LIN {X 0,Y 329.805,Z 667.304,A -85,B 0,C 180,E1 16241.947,E2 16241.947} C_VEL
LIN {X 0,Y 329.564,Z 671.373,A -85,B 0,C 180,E1 16242.444,E2 16242.444} C_VEL
LIN {X 0,Y 319.657,Z 703.267,A -85,B 0,C 180,E1 16245.4,E2 16245.4} C_VEL
LIN {X 0,Y 308.366,Z 732.75,A -85,B 0,C 180,E1 16249.353,E2 16249.353} C_VEL
LIN {X 0,Y 296.702,Z 759.051,A -85,B 0,C 180,E1 16254.413,E2 16254.413} C_VEL
LIN {X 0,Y 286.049,Z 781.446,A -85,B 0,C 180,E1 16260.671,E2 16260.671} C_VEL
LIN {X 0,Y 278.02,Z 798.479,A -85,B 0,C 180,E1 16267.777,E2 16267.777} C_VEL
LIN {X 0,Y 273.133,Z 810.385,A -85,B 0,C 180,E1 16275.599,E2 16275.599} C_VEL
LIN {X 0,Y 271.089,Z 816.889,A -85,B 0,C 180,E1 16283.586,E2 16283.586} C_VEL
LIN {X 0,Y 270.872,Z 818.496,A -85,B 0,C 180,E1 16289.999,E2 16289.999} C_VEL
LIN {X 0,Y 271.134,Z 816.829,A -85,B 0,C 180,E1 16296.412,E2 16296.412} C_VEL
LIN {X 0,Y 273.229,Z 810.161,A -85,B 0,C 180,E1 16304.483,E2 16304.483} C_VEL
LIN {X 0,Y 278.223,Z 797.96,A -85,B 0,C 180,E1 16312.391,E2 16312.391} C_VEL
LIN {X 0,Y 286.286,Z 780.835,A -85,B 0,C 180,E1 16319.419,E2 16319.419} C_VEL
LIN {X 0,Y 296.961,Z 758.345,A -85,B 0,C 180,E1 16325.639,E2 16325.639} C_VEL
LIN {X 0,Y 308.651,Z 731.826,A -85,B 0,C 180,E1 16330.691,E2 16330.691} C_VEL
LIN {X 0,Y 320.1,Z 701.772,A -85,B 0,C 180,E1 16334.662,E2 16334.662} C_VEL
LIN {X 0,Y 330.02,Z 668.599,A -85,B 0,C 180,E1 16337.711,E2 16337.711} C_VEL
LIN {X 0,Y 322.594,Z 643.397,A -85,B 0,C 180,E1 16342.404,E2 16342.404} C_VEL
LIN {X 0,Y 312.412,Z 620.496,A -85,B 0,C 180,E1 16347.568,E2 16347.568} C_VEL
LIN {X 0,Y 300.457,Z 599.556,A -85,B 0,C 180,E1 16353.739,E2 16353.739} C_VEL
LIN {X 0,Y 290.832,Z 585.901,A -85,B 0,C 180,E1 16359.592,E2 16359.592} C_VEL
LIN {X 0,Y 286.331,Z 579.387,A -85,B 0,C 180,E1 16363.177,E2 16363.177} C_VEL
LIN {X 0,Y 282.314,Z 573.377,A -85,B 0,C 180,E1 16367.516,E2 16367.516} C_VEL
LIN {X 0,Y 278.321,Z 569.305,A -85,B 0,C 180,E1 16376.882,E2 16376.882} C_VEL
LIN {X 0,Y 279.401,Z 570.647,A -85,B 0,C 180,E1 16383.301,E2 16383.301} C_VEL
LIN {X 0,Y 282.503,Z 573.483,A -85,B 0,C 180,E1 16388.281,E2 16388.281} C_VEL
LIN {X 0,Y 286.101,Z 579.139,A -85,B 0,C 180,E1 16392.221,E2 16392.221} C_VEL
LIN {X 0,Y 287.999,Z 581.762,A -85,B 0,C 180,E1 16393.861,E2 16393.861} C_VEL
LIN {X 0,Y 293.39,Z 589.45,A -85,B 0,C 180,E1 16397.745,E2 16397.745} C_VEL
LIN {X 0,Y 301.462,Z 601.319,A -85,B 0,C 180,E1 16402.418,E2 16402.418} C_VEL
LIN {X 0,Y 313.146,Z 621.425,A -85,B 0,C 180,E1 16408.222,E2 16408.222} C_VEL
LIN {X 0,Y 323.586,Z 644.854,A -85,B 0,C 180,E1 16413.27,E2 16413.27} C_VEL
LIN {X 0,Y 331.263,Z 670.261,A -85,B 0,C 180,E1 16417.717,E2 16417.717} C_VEL
LIN {X 0,Y 320.897,Z 707.285,A -85,B 0,C 180,E1 16420.726,E2 16420.726} C_VEL
LIN {X 0,Y 309.149,Z 741.143,A -85,B 0,C 180,E1 16424.755,E2 16424.755} C_VEL
LIN {X 0,Y 297.16,Z 771.177,A -85,B 0,C 180,E1 16429.837,E2 16429.837} C_VEL
LIN {X 0,Y 286.1,Z 797.759,A -85,B 0,C 180,E1 16436.244,E2 16436.244} C_VEL
LIN {X 0,Y 277.977,Z 818.25,A -85,B 0,C 180,E1 16443.299,E2 16443.299} C_VEL
LIN {X 0,Y 272.92,Z 834.265,A -85,B 0,C 180,E1 16451.399,E2 16451.399} C_VEL
LIN {X 0,Y 270.979,Z 843.701,A -85,B 0,C 180,E1 16458.924,E2 16458.924} C_VEL
LIN {X 0,Y 270.477,Z 848.401,A -85,B 0,C 180,E1 16466.792,E2 16466.792} C_VEL
LIN {X 0,Y 270.551,Z 848.411,A -85,B 0,C 180,E1 16473.209,E2 16473.209} C_VEL
LIN {X 0,Y 270.986,Z 843.71,A -85,B 0,C 180,E1 16481.085,E2 16481.085} C_VEL
LIN {X 0,Y 273.236,Z 832.973,A -85,B 0,C 180,E1 16489.419,E2 16489.419} C_VEL
LIN {X 0,Y 278.709,Z 816.254,A -85,B 0,C 180,E1 16497.501,E2 16497.501} C_VEL
LIN {X 0,Y 287.215,Z 795.052,A -85,B 0,C 180,E1 16504.52,E2 16504.52} C_VEL
LIN {X 0,Y 297.881,Z 769.444,A -85,B 0,C 180,E1 16510.524,E2 16510.524} C_VEL
LIN {X 0,Y 310.009,Z 738.891,A -85,B 0,C 180,E1 16515.584,E2 16515.584} C_VEL
LIN {X 0,Y 321.936,Z 704.311,A -85,B 0,C 180,E1 16519.579,E2 16519.579} C_VEL
LIN {X 0,Y 331.184,Z 669.723,A -85,B 0,C 180,E1 16522.393,E2 16522.393} C_VEL
LIN {X 0,Y 323.663,Z 644.953,A -85,B 0,C 180,E1 16526.739,E2 16526.739} C_VEL
LIN {X 0,Y 315.532,Z 626.221,A -85,B 0,C 180,E1 16530.694,E2 16530.694} C_VEL
LIN {X 0,Y 311.88,Z 623.31,A -85,B 0,C 180,E1 16532.061,E2 16532.061} C_VEL
LIN {X 0,Y 305.951,Z 620.829,A -85,B 0,C 180,E1 16534.268,E2 16534.268} C_VEL
LIN {X 0,Y 305.532,Z 620.05,A -85,B 0,C 180,E1 16534.493,E2 16534.493} C_VEL
LIN {X 0,Y 295.869,Z 603.458,A -85,B 0,C 180,E1 16539.989,E2 16539.989} C_VEL
LIN {X 0,Y 288.98,Z 593.047,A -85,B 0,C 180,E1 16544.626,E2 16544.626} C_VEL
LIN {X 0,Y 284.687,Z 586.778,A -85,B 0,C 180,E1 16548.302,E2 16548.302} C_VEL
LIN {X 0,Y 281.092,Z 580.621,A -85,B 0,C 180,E1 16552.576,E2 16552.576} C_VEL
LIN {X 0,Y 277.764,Z 577.392,A -85,B 0,C 180,E1 16559.999,E2 16559.999} C_VEL
LIN {X 0,Y 280.92,Z 580.502,A -85,B 0,C 180,E1 16571.484,E2 16571.484} C_VEL
LIN {X 0,Y 284.724,Z 586.915,A -85,B 0,C 180,E1 16576.024,E2 16576.024} C_VEL
LIN {X 0,Y 287.489,Z 591.3,A -85,B 0,C 180,E1 16578.532,E2 16578.532} C_VEL
LIN {X 0,Y 291.493,Z 597.021,A -85,B 0,C 180,E1 16581.518,E2 16581.518} C_VEL
LIN {X 0,Y 299.641,Z 609.825,A -85,B 0,C 180,E1 16586.641,E2 16586.641} C_VEL
LIN {X 0,Y 309.655,Z 628.692,A -85,B 0,C 180,E1 16592.224,E2 16592.224} C_VEL
LIN {X 0,Y 319.03,Z 652.103,A -85,B 0,C 180,E1 16597.568,E2 16597.568} C_VEL
LIN {X 0,Y 324.068,Z 672.936,A -85,B 0,C 180,E1 16601.485,E2 16601.485} C_VEL
LIN {X 0,Y 313.257,Z 706.117,A -85,B 0,C 180,E1 16604.642,E2 16604.642} C_VEL
LIN {X 0,Y 300.569,Z 737.537,A -85,B 0,C 180,E1 16609.072,E2 16609.072} C_VEL
LIN {X 0,Y 287.912,Z 764.286,A -85,B 0,C 180,E1 16614.657,E2 16614.657} C_VEL
LIN {X 0,Y 277.608,Z 784.776,A -85,B 0,C 180,E1 16620.916,E2 16620.916} C_VEL
LIN {X 0,Y 269.758,Z 800.788,A -85,B 0,C 180,E1 16628.163,E2 16628.163} C_VEL
LIN {X 0,Y 264.991,Z 811.989,A -85,B 0,C 180,E1 16636.223,E2 16636.223} C_VEL
LIN {X 0,Y 263.217,Z 817.334,A -85,B 0,C 180,E1 16643.393,E2 16643.393} C_VEL
LIN {X 0,Y 262.982,Z 818.939,A -85,B 0,C 180,E1 16649.999,E2 16649.999} C_VEL
LIN {X 0,Y 263.262,Z 817.274,A -85,B 0,C 180,E1 16656.604,E2 16656.604} C_VEL
LIN {X 0,Y 265.572,Z 810.523,A -85,B 0,C 180,E1 16664.991,E2 16664.991} C_VEL
LIN {X 0,Y 270.838,Z 798.417,A -85,B 0,C 180,E1 16673.036,E2 16673.036} C_VEL
LIN {X 0,Y 279.651,Z 780.628,A -85,B 0,C 180,E1 16680.455,E2 16680.455} C_VEL
LIN {X 0,Y 290.989,Z 757.949,A -85,B 0,C 180,E1 16686.752,E2 16686.752} C_VEL
LIN {X 0,Y 303.284,Z 730.998,A -85,B 0,C 180,E1 16691.888,E2 16691.888} C_VEL
LIN {X 0,Y 315.639,Z 699.335,A -85,B 0,C 180,E1 16696.014,E2 16696.014} C_VEL
LIN {X 0,Y 324.096,Z 671.324,A -85,B 0,C 180,E1 16698.609,E2 16698.609} C_VEL
LIN {X 0,Y 316.842,Z 645.653,A -85,B 0,C 180,E1 16703.659,E2 16703.659} C_VEL
LIN {X 0,Y 306.787,Z 622.65,A -85,B 0,C 180,E1 16709.227,E2 16709.227} C_VEL
LIN {X 0,Y 296.838,Z 605.304,A -85,B 0,C 180,E1 16714.815,E2 16714.815} C_VEL
LIN {X 0,Y 288.776,Z 593.022,A -85,B 0,C 180,E1 16720.224,E2 16720.224} C_VEL
LIN {X 0,Y 284.732,Z 586.895,A -85,B 0,C 180,E1 16723.692,E2 16723.692} C_VEL
LIN {X 0,Y 280.49,Z 580.156,A -85,B 0,C 180,E1 16728.693,E2 16728.693} C_VEL
LIN {X 0,Y 277.532,Z 577.075,A -85,B 0,C 180,E1 16740.001,E2 16740.001} C_VEL
LIN {X 0,Y 281.204,Z 581.256,A -85,B 0,C 180,E1 16747.93,E2 16747.93} C_VEL
LIN {X 0,Y 285.33,Z 587.159,A -85,B 0,C 180,E1 16752.428,E2 16752.428} C_VEL
LIN {X 0,Y 292.338,Z 598.219,A -85,B 0,C 180,E1 16757.908,E2 16757.908} C_VEL
LIN {X 0,Y 301.675,Z 612.953,A -85,B 0,C 180,E1 16763.475,E2 16763.475} C_VEL
LIN {X 0,Y 312.271,Z 633.888,A -85,B 0,C 180,E1 16769.112,E2 16769.112} C_VEL
LIN {X 0,Y 321.29,Z 657.275,A -85,B 0,C 180,E1 16774.026,E2 16774.026} C_VEL
LIN {X 0,Y 325.329,Z 673.89,A -85,B 0,C 180,E1 16776.917,E2 16776.917} C_VEL
LIN {X 0,Y 314.607,Z 709.827,A -85,B 0,C 180,E1 16779.93,E2 16779.93} C_VEL
LIN {X 0,Y 302.053,Z 744.114,A -85,B 0,C 180,E1 16784.161,E2 16784.161} C_VEL
LIN {X 0,Y 289.556,Z 773.856,A -85,B 0,C 180,E1 16789.452,E2 16789.452} C_VEL
LIN {X 0,Y 278.152,Z 799.801,A -85,B 0,C 180,E1 16796.088,E2 16796.088} C_VEL
LIN {X 0,Y 269.934,Z 819.61,A -85,B 0,C 180,E1 16803.339,E2 16803.339} C_VEL
LIN {X 0,Y 265.234,Z 833.802,A -85,B 0,C 180,E1 16810.839,E2 16810.839} C_VEL
LIN {X 0,Y 263.211,Z 842.567,A -85,B 0,C 180,E1 16817.91,E2 16817.91} C_VEL
LIN {X 0,Y 262.653,Z 846.617,A -85,B 0,C 180,E1 16823.38,E2 16823.38} C_VEL
LIN {X 0,Y 262.814,Z 848.446,A -85,B 0,C 180,E1 16830.001,E2 16830.001} C_VEL
LIN {X 0,Y 262.769,Z 845.695,A -85,B 0,C 180,E1 16838.283,E2 16838.283} C_VEL
LIN {X 0,Y 264.269,Z 837.438,A -85,B 0,C 180,E1 16846.647,E2 16846.647} C_VEL
LIN {X 0,Y 268.842,Z 822.671,A -85,B 0,C 180,E1 16855.298,E2 16855.298} C_VEL
LIN {X 0,Y 277.086,Z 802.365,A -85,B 0,C 180,E1 16863.122,E2 16863.122} C_VEL
LIN {X 0,Y 287.795,Z 777.785,A -85,B 0,C 180,E1 16869.701,E2 16869.701} C_VEL
LIN {X 0,Y 299.815,Z 749.596,A -85,B 0,C 180,E1 16875.012,E2 16875.012} C_VEL
LIN {X 0,Y 311.995,Z 717.953,A -85,B 0,C 180,E1 16879.198,E2 16879.198} C_VEL
LIN {X 0,Y 322.866,Z 683.592,A -85,B 0,C 180,E1 16882.382,E2 16882.382} C_VEL
LIN {X 0,Y 325.391,Z 672.786,A -85,B 0,C 180,E1 16883.238,E2 16883.238} C_VEL
LIN {X 0,Y 318.483,Z 648.794,A -85,B 0,C 180,E1 16887.646,E2 16887.646} C_VEL
LIN {X 0,Y 307.903,Z 624.559,A -85,B 0,C 180,E1 16893.242,E2 16893.242} C_VEL
LIN {X 0,Y 305.532,Z 620.05,A -85,B 0,C 180,E1 16894.493,E2 16894.493} C_VEL
LIN {X 0,Y 301.126,Z 615.255,A -85,B 0,C 180,E1 16896.629,E2 16896.629} C_VEL
LIN {X 0,Y 293.286,Z 610.348,A -85,B 0,C 180,E1 16900.537,E2 16900.537} C_VEL
LIN {X 0,Y 286.858,Z 600.102,A -85,B 0,C 180,E1 16905.286,E2 16905.286} C_VEL
LIN {X 0,Y 283.021,Z 594.198,A -85,B 0,C 180,E1 16908.818,E2 16908.818} C_VEL
LIN {X 0,Y 279.274,Z 587.733,A -85,B 0,C 180,E1 16913.775,E2 16913.775} C_VEL
LIN {X 0,Y 276.799,Z 585.255,A -85,B 0,C 180,E1 16919.999,E2 16919.999} C_VEL
LIN {X 0,Y 279.653,Z 588.2,A -85,B 0,C 180,E1 16931.09,E2 16931.09} C_VEL
LIN {X 0,Y 283.599,Z 594.784,A -85,B 0,C 180,E1 16936.034,E2 16936.034} C_VEL
LIN {X 0,Y 289.739,Z 604.964,A -85,B 0,C 180,E1 16941.354,E2 16941.354} C_VEL
LIN {X 0,Y 298.315,Z 619.221,A -85,B 0,C 180,E1 16947.075,E2 16947.075} C_VEL
LIN {X 0,Y 308.334,Z 640.87,A -85,B 0,C 180,E1 16953.193,E2 16953.193} C_VEL
LIN {X 0,Y 316.21,Z 664.666,A -85,B 0,C 180,E1 16958.492,E2 16958.492} C_VEL
LIN {X 0,Y 318.119,Z 676.365,A -85,B 0,C 180,E1 16960.637,E2 16960.637} C_VEL
LIN {X 0,Y 306.215,Z 710.801,A -85,B 0,C 180,E1 16964.082,E2 16964.082} C_VEL
LIN {X 0,Y 293.721,Z 739.941,A -85,B 0,C 180,E1 16968.404,E2 16968.404} C_VEL
LIN {X 0,Y 281.094,Z 765.428,A -85,B 0,C 180,E1 16973.889,E2 16973.889} C_VEL
LIN {X 0,Y 269.837,Z 786.779,A -85,B 0,C 180,E1 16980.676,E2 16980.676} C_VEL
LIN {X 0,Y 261.563,Z 802.907,A -85,B 0,C 180,E1 16988.467,E2 16988.467} C_VEL
LIN {X 0,Y 257.087,Z 813.025,A -85,B 0,C 180,E1 16996.374,E2 16996.374} C_VEL
LIN {X 0,Y 255.348,Z 817.779,A -85,B 0,C 180,E1 17003.189,E2 17003.189} C_VEL
LIN {X 0,Y 255.104,Z 819.381,A -85,B 0,C 180,E1 17009.999,E2 17009.999} C_VEL
LIN {X 0,Y 255.393,Z 817.719,A -85,B 0,C 180,E1 17016.809,E2 17016.809} C_VEL
LIN {X 0,Y 257.816,Z 811.109,A -85,B 0,C 180,E1 17025.323,E2 17025.323} C_VEL
LIN {X 0,Y 263.481,Z 798.875,A -85,B 0,C 180,E1 17033.718,E2 17033.718} C_VEL
LIN {X 0,Y 272.843,Z 780.982,A -85,B 0,C 180,E1 17041.347,E2 17041.347} C_VEL
LIN {X 0,Y 284.656,Z 758.446,A -85,B 0,C 180,E1 17047.71,E2 17047.71} C_VEL
LIN {X 0,Y 297.417,Z 731.526,A -85,B 0,C 180,E1 17052.911,E2 17052.911} C_VEL
LIN {X 0,Y 310.208,Z 699.948,A -85,B 0,C 180,E1 17057.063,E2 17057.063} C_VEL
LIN {X 0,Y 318.212,Z 675.713,A -85,B 0,C 180,E1 17059.307,E2 17059.307} C_VEL
LIN {X 0,Y 313.01,Z 653.846,A -85,B 0,C 180,E1 17063.666,E2 17063.666} C_VEL
LIN {X 0,Y 304.503,Z 632.045,A -85,B 0,C 180,E1 17068.971,E2 17068.971} C_VEL
LIN {X 0,Y 294.728,Z 612.975,A -85,B 0,C 180,E1 17075.028,E2 17075.028} C_VEL
LIN {X 0,Y 286.754,Z 600.077,A -85,B 0,C 180,E1 17080.833,E2 17080.833} C_VEL
LIN {X 0,Y 282.911,Z 594.239,A -85,B 0,C 180,E1 17084.322,E2 17084.322} C_VEL
LIN {X 0,Y 279.15,Z 587.803,A -85,B 0,C 180,E1 17089.22,E2 17089.22} C_VEL
LIN {X 0,Y 276.565,Z 584.949,A -85,B 0,C 180,E1 17100.001,E2 17100.001} C_VEL
LIN {X 0,Y 279.914,Z 588.926,A -85,B 0,C 180,E1 17107.558,E2 17107.558} C_VEL
LIN {X 0,Y 284.911,Z 597.129,A -85,B 0,C 180,E1 17113.202,E2 17113.202} C_VEL
LIN {X 0,Y 289.868,Z 604.891,A -85,B 0,C 180,E1 17117.183,E2 17117.183} C_VEL
LIN {X 0,Y 298.813,Z 619.998,A -85,B 0,C 180,E1 17123.022,E2 17123.022} C_VEL
LIN {X 0,Y 308.473,Z 640.294,A -85,B 0,C 180,E1 17128.619,E2 17128.619} C_VEL
LIN {X 0,Y 316.841,Z 664.054,A -85,B 0,C 180,E1 17133.744,E2 17133.744} C_VEL
LIN {X 0,Y 319.486,Z 677.138,A -85,B 0,C 180,E1 17136.043,E2 17136.043} C_VEL
LIN {X 0,Y 307.678,Z 714.335,A -85,B 0,C 180,E1 17139.314,E2 17139.314} C_VEL
LIN {X 0,Y 294.546,Z 747.936,A -85,B 0,C 180,E1 17143.71,E2 17143.71} C_VEL
LIN {X 0,Y 281.914,Z 776.391,A -85,B 0,C 180,E1 17149.056,E2 17149.056} C_VEL
LIN {X 0,Y 270.757,Z 800.612,A -85,B 0,C 180,E1 17155.536,E2 17155.536} C_VEL
LIN {X 0,Y 262.182,Z 820.21,A -85,B 0,C 180,E1 17163.033,E2 17163.033} C_VEL
LIN {X 0,Y 257.043,Z 835.072,A -85,B 0,C 180,E1 17171.469,E2 17171.469} C_VEL
LIN {X 0,Y 255.053,Z 843.972,A -85,B 0,C 180,E1 17179.742,E2 17179.742} C_VEL
LIN {X 0,Y 254.688,Z 847.513,A -85,B 0,C 180,E1 17186.593,E2 17186.593} C_VEL
LIN {X 0,Y 254.918,Z 848.003,A -85,B 0,C 180,E1 17190.001,E2 17190.001} C_VEL
LIN {X 0,Y 254.767,Z 846.182,A -85,B 0,C 180,E1 17196.827,E2 17196.827} C_VEL
LIN {X 0,Y 256.035,Z 839.046,A -85,B 0,C 180,E1 17205.433,E2 17205.433} C_VEL
LIN {X 0,Y 259.94,Z 826.104,A -85,B 0,C 180,E1 17214.063,E2 17214.063} C_VEL
LIN {X 0,Y 267.767,Z 807.41,A -85,B 0,C 180,E1 17222.177,E2 17222.177} C_VEL
LIN {X 0,Y 278.559,Z 783.894,A -85,B 0,C 180,E1 17229.188,E2 17229.188} C_VEL
LIN {X 0,Y 291.796,Z 754.474,A -85,B 0,C 180,E1 17235.263,E2 17235.263} C_VEL
LIN {X 0,Y 304.992,Z 722.106,A -85,B 0,C 180,E1 17239.811,E2 17239.811} C_VEL
LIN {X 0,Y 316.525,Z 687.743,A -85,B 0,C 180,E1 17243.166,E2 17243.166} C_VEL
LIN {X 0,Y 319.637,Z 675.715,A -85,B 0,C 180,E1 17244.14,E2 17244.14} C_VEL
LIN {X 0,Y 313.177,Z 652.194,A -85,B 0,C 180,E1 17248.689,E2 17248.689} C_VEL
LIN {X 0,Y 303.011,Z 628.055,A -85,B 0,C 180,E1 17254.609,E2 17254.609} C_VEL
LIN {X 0,Y 293.611,Z 610.921,A -85,B 0,C 180,E1 17260.319,E2 17260.319} C_VEL
LIN {X 0,Y 293.286,Z 610.348,A -85,B 0,C 180,E1 17260.537,E2 17260.537} C_VEL
LIN {X 0,Y 289.279,Z 607.619,A -85,B 0,C 180,E1 17262.952,E2 17262.952} C_VEL
LIN {X 0,Y 283.72,Z 605.63,A -85,B 0,C 180,E1 17266.774,E2 17266.774} C_VEL
LIN {X 0,Y 283.308,Z 604.905,A -85,B 0,C 180,E1 17267.189,E2 17267.189} C_VEL
LIN {X 0,Y 280.815,Z 601.071,A -85,B 0,C 180,E1 17269.859,E2 17269.859} C_VEL
LIN {X 0,Y 277.923,Z 595.442,A -85,B 0,C 180,E1 17274.137,E2 17274.137} C_VEL
LIN {X 0,Y 275.75,Z 593.111,A -85,B 0,C 180,E1 17279.999,E2 17279.999} C_VEL
LIN {X 0,Y 278.293,Z 595.941,A -85,B 0,C 180,E1 17290.772,E2 17290.772} C_VEL
LIN {X 0,Y 283.105,Z 604.787,A -85,B 0,C 180,E1 17296.992,E2 17296.992} C_VEL
LIN {X 0,Y 289.531,Z 615.273,A -85,B 0,C 180,E1 17302.48,E2 17302.48} C_VEL
LIN {X 0,Y 298.618,Z 633.439,A -85,B 0,C 180,E1 17308.901,E2 17308.901} C_VEL
LIN {X 0,Y 306.776,Z 654.417,A -85,B 0,C 180,E1 17314.491,E2 17314.491} C_VEL
LIN {X 0,Y 312.579,Z 677.351,A -85,B 0,C 180,E1 17319.471,E2 17319.471} C_VEL
LIN {X 0,Y 300.494,Z 712.018,A -85,B 0,C 180,E1 17323.083,E2 17323.083} C_VEL
LIN {X 0,Y 287.425,Z 741.295,A -85,B 0,C 180,E1 17327.511,E2 17327.511} C_VEL
LIN {X 0,Y 275.049,Z 765.249,A -85,B 0,C 180,E1 17332.733,E2 17332.733} C_VEL
LIN {X 0,Y 263.124,Z 786.826,A -85,B 0,C 180,E1 17339.661,E2 17339.661} C_VEL
LIN {X 0,Y 254.007,Z 803.629,A -85,B 0,C 180,E1 17347.987,E2 17347.987} C_VEL
LIN {X 0,Y 249.141,Z 813.914,A -85,B 0,C 180,E1 17356.471,E2 17356.471} C_VEL
LIN {X 0,Y 247.482,Z 818.223,A -85,B 0,C 180,E1 17362.971,E2 17362.971} C_VEL
LIN {X 0,Y 247.214,Z 819.824,A -85,B 0,C 180,E1 17369.999,E2 17369.999} C_VEL
LIN {X 0,Y 247.526,Z 818.165,A -85,B 0,C 180,E1 17377.026,E2 17377.026} C_VEL
LIN {X 0,Y 250.129,Z 811.56,A -85,B 0,C 180,E1 17385.806,E2 17385.806} C_VEL
LIN {X 0,Y 256.168,Z 799.331,A -85,B 0,C 180,E1 17394.438,E2 17394.438} C_VEL
LIN {X 0,Y 266.053,Z 781.457,A -85,B 0,C 180,E1 17402.242,E2 17402.242} C_VEL
LIN {X 0,Y 278.385,Z 758.942,A -85,B 0,C 180,E1 17408.714,E2 17408.714} C_VEL
LIN {X 0,Y 291.672,Z 732.057,A -85,B 0,C 180,E1 17413.97,E2 17413.97} C_VEL
LIN {X 0,Y 304.9,Z 700.549,A -85,B 0,C 180,E1 17418.146,E2 17418.146} C_VEL
LIN {X 0,Y 312.476,Z 678.562,A -85,B 0,C 180,E1 17420.239,E2 17420.239} C_VEL
LIN {X 0,Y 307.732,Z 657.363,A -85,B 0,C 180,E1 17424.686,E2 17424.686} C_VEL
LIN {X 0,Y 299.64,Z 635.657,A -85,B 0,C 180,E1 17430.272,E2 17430.272} C_VEL
LIN {X 0,Y 291.027,Z 618.526,A -85,B 0,C 180,E1 17436.123,E2 17436.123} C_VEL
LIN {X 0,Y 284.307,Z 606.939,A -85,B 0,C 180,E1 17441.569,E2 17441.569} C_VEL
LIN {X 0,Y 281.302,Z 601.772,A -85,B 0,C 180,E1 17444.687,E2 17444.687} C_VEL
LIN {X 0,Y 277.671,Z 595.48,A -85,B 0,C 180,E1 17449.745,E2 17449.745} C_VEL
LIN {X 0,Y 275.523,Z 592.805,A -85,B 0,C 180,E1 17460.001,E2 17460.001} C_VEL
LIN {X 0,Y 278.545,Z 596.738,A -85,B 0,C 180,E1 17467.282,E2 17467.282} C_VEL
LIN {X 0,Y 283.097,Z 604.545,A -85,B 0,C 180,E1 17472.768,E2 17472.768} C_VEL
LIN {X 0,Y 289.707,Z 615.313,A -85,B 0,C 180,E1 17478.274,E2 17478.274} C_VEL
LIN {X 0,Y 298.97,Z 633.723,A -85,B 0,C 180,E1 17484.636,E2 17484.636} C_VEL
LIN {X 0,Y 307.826,Z 655.658,A -85,B 0,C 180,E1 17490.273,E2 17490.273} C_VEL
LIN {X 0,Y 313.866,Z 678.411,A -85,B 0,C 180,E1 17494.91,E2 17494.91} C_VEL
LIN {X 0,Y 302.227,Z 714.704,A -85,B 0,C 180,E1 17498.238,E2 17498.238} C_VEL
LIN {X 0,Y 288.952,Z 747.376,A -85,B 0,C 180,E1 17502.537,E2 17502.537} C_VEL
LIN {X 0,Y 275.775,Z 775.875,A -85,B 0,C 180,E1 17507.94,E2 17507.94} C_VEL
LIN {X 0,Y 264.374,Z 799.404,A -85,B 0,C 180,E1 17514.293,E2 17514.293} C_VEL
LIN {X 0,Y 254.913,Z 819.719,A -85,B 0,C 180,E1 17522.19,E2 17522.19} C_VEL
LIN {X 0,Y 249.308,Z 834.779,A -85,B 0,C 180,E1 17530.999,E2 17530.999} C_VEL
LIN {X 0,Y 247.177,Z 843.521,A -85,B 0,C 180,E1 17539.412,E2 17539.412} C_VEL
LIN {X 0,Y 246.785,Z 847.068,A -85,B 0,C 180,E1 17546.483,E2 17546.483} C_VEL
LIN {X 0,Y 247.023,Z 847.56,A -85,B 0,C 180,E1 17550.001,E2 17550.001} C_VEL
LIN {X 0,Y 246.878,Z 845.735,A -85,B 0,C 180,E1 17557.046,E2 17557.046} C_VEL
LIN {X 0,Y 247.81,Z 840.474,A -85,B 0,C 180,E1 17564.146,E2 17564.146} C_VEL
LIN {X 0,Y 251.344,Z 828.737,A -85,B 0,C 180,E1 17573.052,E2 17573.052} C_VEL
LIN {X 0,Y 259.117,Z 810.719,A -85,B 0,C 180,E1 17581.728,E2 17581.728} C_VEL
LIN {X 0,Y 270.089,Z 787.935,A -85,B 0,C 180,E1 17589.099,E2 17589.099} C_VEL
LIN {X 0,Y 283.221,Z 760.281,A -85,B 0,C 180,E1 17595.271,E2 17595.271} C_VEL
LIN {X 0,Y 296.486,Z 729.708,A -85,B 0,C 180,E1 17599.997,E2 17599.997} C_VEL
LIN {X 0,Y 309.019,Z 695.526,A -85,B 0,C 180,E1 17603.642,E2 17603.642} C_VEL
LIN {X 0,Y 313.994,Z 678.693,A -85,B 0,C 180,E1 17605.058,E2 17605.058} C_VEL
LIN {X 0,Y 307.426,Z 654.193,A -85,B 0,C 180,E1 17610.091,E2 17610.091} C_VEL
LIN {X 0,Y 297.825,Z 630.835,A -85,B 0,C 180,E1 17616.237,E2 17616.237} C_VEL
LIN {X 0,Y 288.817,Z 613.865,A -85,B 0,C 180,E1 17622.485,E2 17622.485} C_VEL
LIN {X 0,Y 283.308,Z 604.905,A -85,B 0,C 180,E1 17627.189,E2 17627.189} C_VEL
LIN {X 0,Y 280.708,Z 602.633,A -85,B 0,C 180,E1 17629.73,E2 17629.73} C_VEL
LIN {X 0,Y 276.668,Z 603.213,A -85,B 0,C 180,E1 17634.206,E2 17634.206} C_VEL
LIN {X 0,Y 274.599,Z 600.951,A -85,B 0,C 180,E1 17639.999,E2 17639.999} C_VEL
LIN {X 0,Y 276.817,Z 603.8,A -85,B 0,C 180,E1 17650.525,E2 17650.525} C_VEL
LIN {X 0,Y 281.412,Z 612.742,A -85,B 0,C 180,E1 17656.908,E2 17656.908} C_VEL
LIN {X 0,Y 287.157,Z 623.101,A -85,B 0,C 180,E1 17662.267,E2 17662.267} C_VEL
LIN {X 0,Y 294.92,Z 639.795,A -85,B 0,C 180,E1 17668.349,E2 17668.349} C_VEL
LIN {X 0,Y 302.125,Z 659.9,A -85,B 0,C 180,E1 17673.88,E2 17673.88} C_VEL
LIN {X 0,Y 306.803,Z 679.959,A -85,B 0,C 180,E1 17678.439,E2 17678.439} C_VEL
LIN {X 0,Y 305.106,Z 686.647,A -85,B 0,C 180,E1 17679.183,E2 17679.183} C_VEL
LIN {X 0,Y 292.269,Z 719.29,A -85,B 0,C 180,E1 17682.826,E2 17682.826} C_VEL
LIN {X 0,Y 278.061,Z 748.706,A -85,B 0,C 180,E1 17687.747,E2 17687.747} C_VEL
LIN {X 0,Y 264.812,Z 772.632,A -85,B 0,C 180,E1 17693.656,E2 17693.656} C_VEL
LIN {X 0,Y 253.437,Z 792.036,A -85,B 0,C 180,E1 17700.794,E2 17700.794} C_VEL
LIN {X 0,Y 245.13,Z 806.813,A -85,B 0,C 180,E1 17709.197,E2 17709.197} C_VEL
LIN {X 0,Y 240.807,Z 815.796,A -85,B 0,C 180,E1 17717.8,E2 17717.8} C_VEL
LIN {X 0,Y 239.278,Z 819.858,A -85,B 0,C 180,E1 17726.371,E2 17726.371} C_VEL
LIN {X 0,Y 239.374,Z 819.82,A -85,B 0,C 180,E1 17733.626,E2 17733.626} C_VEL
LIN {X 0,Y 240.884,Z 815.652,A -85,B 0,C 180,E1 17742.247,E2 17742.247} C_VEL
LIN {X 0,Y 245.852,Z 805.379,A -85,B 0,C 180,E1 17751.684,E2 17751.684} C_VEL
LIN {X 0,Y 255.179,Z 789.097,A -85,B 0,C 180,E1 17760.399,E2 17760.399} C_VEL
LIN {X 0,Y 267.794,Z 767.327,A -85,B 0,C 180,E1 17767.747,E2 17767.747} C_VEL
LIN {X 0,Y 281.531,Z 741.717,A -85,B 0,C 180,E1 17773.494,E2 17773.494} C_VEL
LIN {X 0,Y 295.374,Z 711.857,A -85,B 0,C 180,E1 17778.018,E2 17778.018} C_VEL
LIN {X 0,Y 306.881,Z 681.089,A -85,B 0,C 180,E1 17781.206,E2 17781.206} C_VEL
LIN {X 0,Y 301.546,Z 657.866,A -85,B 0,C 180,E1 17786.478,E2 17786.478} C_VEL
LIN {X 0,Y 293.776,Z 636.988,A -85,B 0,C 180,E1 17792.368,E2 17792.368} C_VEL
LIN {X 0,Y 285.758,Z 620.759,A -85,B 0,C 180,E1 17798.64,E2 17798.64} C_VEL
LIN {X 0,Y 279.752,Z 609.582,A -85,B 0,C 180,E1 17804.704,E2 17804.704} C_VEL
LIN {X 0,Y 276.191,Z 603.167,A -85,B 0,C 180,E1 17810.113,E2 17810.113} C_VEL
LIN {X 0,Y 274.373,Z 600.644,A -85,B 0,C 180,E1 17820.001,E2 17820.001} C_VEL
LIN {X 0,Y 277.005,Z 604.345,A -85,B 0,C 180,E1 17826.904,E2 17826.904} C_VEL
LIN {X 0,Y 281.342,Z 612.428,A -85,B 0,C 180,E1 17832.64,E2 17832.64} C_VEL
LIN {X 0,Y 287.176,Z 622.801,A -85,B 0,C 180,E1 17837.944,E2 17837.944} C_VEL
LIN {X 0,Y 295.591,Z 640.509,A -85,B 0,C 180,E1 17844.189,E2 17844.189} C_VEL
LIN {X 0,Y 303.55,Z 662.268,A -85,B 0,C 180,E1 17849.918,E2 17849.918} C_VEL
LIN {X 0,Y 308.108,Z 682.705,A -85,B 0,C 180,E1 17854.159,E2 17854.159} C_VEL
LIN {X 0,Y 295.883,Z 717.549,A -85,B 0,C 180,E1 17857.395,E2 17857.395} C_VEL
LIN {X 0,Y 282.093,Z 749.926,A -85,B 0,C 180,E1 17861.831,E2 17861.831} C_VEL
LIN {X 0,Y 267.578,Z 779.69,A -85,B 0,C 180,E1 17867.785,E2 17867.785} C_VEL
LIN {X 0,Y 254.905,Z 804.508,A -85,B 0,C 180,E1 17875.134,E2 17875.134} C_VEL
LIN {X 0,Y 245.787,Z 823.55,A -85,B 0,C 180,E1 17883.503,E2 17883.503} C_VEL
LIN {X 0,Y 240.767,Z 837.077,A -85,B 0,C 180,E1 17892.621,E2 17892.621} C_VEL
LIN {X 0,Y 239.138,Z 844.34,A -85,B 0,C 180,E1 17900.894,E2 17900.894} C_VEL
LIN {X 0,Y 239.138,Z 847.117,A -85,B 0,C 180,E1 17910.001,E2 17910.001} C_VEL
LIN {X 0,Y 239.002,Z 845.29,A -85,B 0,C 180,E1 17917.279,E2 17917.279} C_VEL
LIN {X 0,Y 240,Z 840.02,A -85,B 0,C 180,E1 17924.617,E2 17924.617} C_VEL
LIN {X 0,Y 243.831,Z 828.272,A -85,B 0,C 180,E1 17933.805,E2 17933.805} C_VEL
LIN {X 0,Y 252.353,Z 809.829,A -85,B 0,C 180,E1 17942.869,E2 17942.869} C_VEL
LIN {X 0,Y 264.467,Z 785.915,A -85,B 0,C 180,E1 17950.634,E2 17950.634} C_VEL
LIN {X 0,Y 277.89,Z 758.907,A -85,B 0,C 180,E1 17956.632,E2 17956.632} C_VEL
LIN {X 0,Y 291.908,Z 727.704,A -85,B 0,C 180,E1 17961.404,E2 17961.404} C_VEL
LIN {X 0,Y 305.079,Z 692.579,A -85,B 0,C 180,E1 17965.063,E2 17965.063} C_VEL
LIN {X 0,Y 308.313,Z 682,A -85,B 0,C 180,E1 17965.94,E2 17965.94} C_VEL
LIN {X 0,Y 302.688,Z 659.287,A -85,B 0,C 180,E1 17970.812,E2 17970.812} C_VEL
LIN {X 0,Y 294.115,Z 636.852,A -85,B 0,C 180,E1 17976.95,E2 17976.95} C_VEL
LIN {X 0,Y 286.145,Z 620.801,A -85,B 0,C 180,E1 17983.036,E2 17983.036} C_VEL
LIN {X 0,Y 279.917,Z 609.543,A -85,B 0,C 180,E1 17989.198,E2 17989.198} C_VEL
LIN {X 0,Y 276.668,Z 603.213,A -85,B 0,C 180,E1 17994.206,E2 17994.206} C_VEL
LIN {X 0,Y 274.312,Z 605.745,A -85,B 0,C 180,E1 17997.788,E2 17997.788} C_VEL
LIN {X 0,Y 272.952,Z 608.751,A -85,B 0,C 180,E1 18001.419,E2 18001.419} C_VEL
LIN {X 0,Y 275.258,Z 612.102,A -85,B 0,C 180,E1 18010.597,E2 18010.597} C_VEL
LIN {X 0,Y 279.146,Z 620.07,A -85,B 0,C 180,E1 18016.542,E2 18016.542} C_VEL
LIN {X 0,Y 284.668,Z 631.133,A -85,B 0,C 180,E1 18022.218,E2 18022.218} C_VEL
LIN {X 0,Y 292.034,Z 648.241,A -85,B 0,C 180,E1 18028.487,E2 18028.487} C_VEL
LIN {X 0,Y 298.429,Z 669.224,A -85,B 0,C 180,E1 18034.238,E2 18034.238} C_VEL
LIN {X 0,Y 300.994,Z 685.004,A -85,B 0,C 180,E1 18037.811,E2 18037.811} C_VEL
LIN {X 0,Y 287.77,Z 718.028,A -85,B 0,C 180,E1 18041.434,E2 18041.434} C_VEL
LIN {X 0,Y 273.443,Z 747.036,A -85,B 0,C 180,E1 18046.172,E2 18046.172} C_VEL
LIN {X 0,Y 259.026,Z 772.118,A -85,B 0,C 180,E1 18052.303,E2 18052.303} C_VEL
LIN {X 0,Y 246.96,Z 791.729,A -85,B 0,C 180,E1 18059.533,E2 18059.533} C_VEL
LIN {X 0,Y 238.377,Z 805.994,A -85,B 0,C 180,E1 18067.598,E2 18067.598} C_VEL
LIN {X 0,Y 233.224,Z 815.805,A -85,B 0,C 180,E1 18076.829,E2 18076.829} C_VEL
LIN {X 0,Y 231.389,Z 820.302,A -85,B 0,C 180,E1 18086.248,E2 18086.248} C_VEL
LIN {X 0,Y 231.484,Z 820.264,A -85,B 0,C 180,E1 18093.749,E2 18093.749} C_VEL
LIN {X 0,Y 233.329,Z 815.615,A -85,B 0,C 180,E1 18103.281,E2 18103.281} C_VEL
LIN {X 0,Y 238.449,Z 805.833,A -85,B 0,C 180,E1 18112.393,E2 18112.393} C_VEL
LIN {X 0,Y 248.024,Z 790.02,A -85,B 0,C 180,E1 18121.122,E2 18121.122} C_VEL
LIN {X 0,Y 261.157,Z 768.467,A -85,B 0,C 180,E1 18128.637,E2 18128.637} C_VEL
LIN {X 0,Y 275.592,Z 742.687,A -85,B 0,C 180,E1 18134.543,E2 18134.543} C_VEL
LIN {X 0,Y 289.398,Z 714.139,A -85,B 0,C 180,E1 18138.955,E2 18138.955} C_VEL
LIN {X 0,Y 301.083,Z 683.583,A -85,B 0,C 180,E1 18142.287,E2 18142.287} C_VEL
LIN {X 0,Y 295.948,Z 660.094,A -85,B 0,C 180,E1 18147.945,E2 18147.945} C_VEL
LIN {X 0,Y 288.405,Z 639.309,A -85,B 0,C 180,E1 18154.337,E2 18154.337} C_VEL
LIN {X 0,Y 280.803,Z 622.937,A -85,B 0,C 180,E1 18161.432,E2 18161.432} C_VEL
LIN {X 0,Y 276.872,Z 616.072,A -85,B 0,C 180,E1 18166.059,E2 18166.059} C_VEL
LIN {X 0,Y 274.493,Z 610.764,A -85,B 0,C 180,E1 18170.476,E2 18170.476} C_VEL
LIN {X 0,Y 272.919,Z 608.423,A -85,B 0,C 180,E1 18180.001,E2 18180.001} C_VEL
LIN {X 0,Y 275.293,Z 612.017,A -85,B 0,C 180,E1 18186.631,E2 18186.631} C_VEL
LIN {X 0,Y 279.279,Z 620.104,A -85,B 0,C 180,E1 18192.424,E2 18192.424} C_VEL
LIN {X 0,Y 284.653,Z 630.439,A -85,B 0,C 180,E1 18197.708,E2 18197.708} C_VEL
LIN {X 0,Y 291.907,Z 647.036,A -85,B 0,C 180,E1 18203.7,E2 18203.7} C_VEL
LIN {X 0,Y 299.167,Z 668.731,A -85,B 0,C 180,E1 18209.548,E2 18209.548} C_VEL
LIN {X 0,Y 302.398,Z 685.789,A -85,B 0,C 180,E1 18213.187,E2 18213.187} C_VEL
LIN {X 0,Y 289.164,Z 721.556,A -85,B 0,C 180,E1 18216.654,E2 18216.654} C_VEL
LIN {X 0,Y 273.861,Z 755.21,A -85,B 0,C 180,E1 18221.559,E2 18221.559} C_VEL
LIN {X 0,Y 259.056,Z 783.81,A -85,B 0,C 180,E1 18227.77,E2 18227.77} C_VEL
LIN {X 0,Y 246.974,Z 806.29,A -85,B 0,C 180,E1 18234.92,E2 18234.92} C_VEL
LIN {X 0,Y 237.726,Z 824.655,A -85,B 0,C 180,E1 18243.525,E2 18243.525} C_VEL
LIN {X 0,Y 232.729,Z 837.649,A -85,B 0,C 180,E1 18252.978,E2 18252.978} C_VEL
LIN {X 0,Y 231.259,Z 843.934,A -85,B 0,C 180,E1 18260.665,E2 18260.665} C_VEL
LIN {X 0,Y 231.241,Z 846.674,A -85,B 0,C 180,E1 18270.001,E2 18270.001} C_VEL
LIN {X 0,Y 231.114,Z 844.843,A -85,B 0,C 180,E1 18277.529,E2 18277.529} C_VEL
LIN {X 0,Y 232.203,Z 839.566,A -85,B 0,C 180,E1 18285.119,E2 18285.119} C_VEL
LIN {X 0,Y 236.368,Z 827.807,A -85,B 0,C 180,E1 18294.606,E2 18294.606} C_VEL
LIN {X 0,Y 245.289,Z 809.758,A -85,B 0,C 180,E1 18303.748,E2 18303.748} C_VEL
LIN {X 0,Y 257.491,Z 786.926,A -85,B 0,C 180,E1 18311.415,E2 18311.415} C_VEL
LIN {X 0,Y 271.729,Z 759.583,A -85,B 0,C 180,E1 18317.661,E2 18317.661} C_VEL
LIN {X 0,Y 286.298,Z 728.53,A -85,B 0,C 180,E1 18322.492,E2 18322.492} C_VEL
LIN {X 0,Y 299.681,Z 694.233,A -85,B 0,C 180,E1 18326.127,E2 18326.127} C_VEL
LIN {X 0,Y 302.558,Z 684.453,A -85,B 0,C 180,E1 18327.032,E2 18327.032} C_VEL
LIN {X 0,Y 297.241,Z 662.082,A -85,B 0,C 180,E1 18332.143,E2 18332.143} C_VEL
LIN {X 0,Y 290.215,Z 642.607,A -85,B 0,C 180,E1 18337.777,E2 18337.777} C_VEL
LIN {X 0,Y 283.322,Z 627.534,A -85,B 0,C 180,E1 18343.684,E2 18343.684} C_VEL
LIN {X 0,Y 277.758,Z 616.883,A -85,B 0,C 180,E1 18349.746,E2 18349.746} C_VEL
LIN {X 0,Y 274.763,Z 610.789,A -85,B 0,C 180,E1 18354.862,E2 18354.862} C_VEL
LIN {X 0,Y 272.952,Z 608.751,A -85,B 0,C 180,E1 18361.419,E2 18361.419} C_VEL
LIN {X 0,Y 272.566,Z 611.542,A -85,B 0,C 180,E1 18364.11,E2 18364.11} C_VEL
LIN {X 0,Y 272.533,Z 618.307,A -85,B 0,C 180,E1 18368.53,E2 18368.53} C_VEL
LIN {X 0,Y 273.678,Z 621.179,A -85,B 0,C 180,E1 18371.365,E2 18371.365} C_VEL
LIN {X 0,Y 276.754,Z 627.427,A -85,B 0,C 180,E1 18376.179,E2 18376.179} C_VEL
LIN {X 0,Y 281.408,Z 637.429,A -85,B 0,C 180,E1 18381.495,E2 18381.495} C_VEL
LIN {X 0,Y 287.888,Z 654.094,A -85,B 0,C 180,E1 18387.82,E2 18387.82} C_VEL
LIN {X 0,Y 293.337,Z 673.899,A -85,B 0,C 180,E1 18393.481,E2 18393.481} C_VEL
LIN {X 0,Y 295.493,Z 687.731,A -85,B 0,C 180,E1 18396.793,E2 18396.793} C_VEL
LIN {X 0,Y 281.065,Z 721.772,A -85,B 0,C 180,E1 18400.657,E2 18400.657} C_VEL
LIN {X 0,Y 266.763,Z 749.271,A -85,B 0,C 180,E1 18405.36,E2 18405.36} C_VEL
LIN {X 0,Y 252.351,Z 773.228,A -85,B 0,C 180,E1 18411.397,E2 18411.397} C_VEL
LIN {X 0,Y 239.437,Z 793.199,A -85,B 0,C 180,E1 18419.041,E2 18419.041} C_VEL
LIN {X 0,Y 230.273,Z 807.716,A -85,B 0,C 180,E1 18427.785,E2 18427.785} C_VEL
LIN {X 0,Y 225.481,Z 816.251,A -85,B 0,C 180,E1 18436.368,E2 18436.368} C_VEL
LIN {X 0,Y 223.501,Z 820.745,A -85,B 0,C 180,E1 18446.115,E2 18446.115} C_VEL
LIN {X 0,Y 223.594,Z 820.708,A -85,B 0,C 180,E1 18453.882,E2 18453.882} C_VEL
LIN {X 0,Y 225.586,Z 816.063,A -85,B 0,C 180,E1 18463.745,E2 18463.745} C_VEL
LIN {X 0,Y 231.064,Z 806.286,A -85,B 0,C 180,E1 18473.15,E2 18473.15} C_VEL
LIN {X 0,Y 241.054,Z 790.737,A -85,B 0,C 180,E1 18481.981,E2 18481.981} C_VEL
LIN {X 0,Y 254.623,Z 769.525,A -85,B 0,C 180,E1 18489.598,E2 18489.598} C_VEL
LIN {X 0,Y 269.777,Z 743.568,A -85,B 0,C 180,E1 18495.659,E2 18495.659} C_VEL
LIN {X 0,Y 284.077,Z 715.128,A -85,B 0,C 180,E1 18500.103,E2 18500.103} C_VEL
LIN {X 0,Y 295.438,Z 686.693,A -85,B 0,C 180,E1 18503.278,E2 18503.278} C_VEL
LIN {X 0,Y 291.245,Z 665.241,A -85,B 0,C 180,E1 18508.681,E2 18508.681} C_VEL
LIN {X 0,Y 284.909,Z 645.927,A -85,B 0,C 180,E1 18514.843,E2 18514.843} C_VEL
LIN {X 0,Y 277.866,Z 629.682,A -85,B 0,C 180,E1 18522.154,E2 18522.154} C_VEL
LIN {X 0,Y 274.56,Z 623.212,A -85,B 0,C 180,E1 18526.65,E2 18526.65} C_VEL
LIN {X 0,Y 272.571,Z 618.379,A -85,B 0,C 180,E1 18530.812,E2 18530.812} C_VEL
LIN {X 0,Y 271.324,Z 616.146,A -85,B 0,C 180,E1 18540.001,E2 18540.001} C_VEL
LIN {X 0,Y 273.355,Z 619.649,A -85,B 0,C 180,E1 18546.36,E2 18546.36} C_VEL
LIN {X 0,Y 277.097,Z 627.757,A -85,B 0,C 180,E1 18552.223,E2 18552.223} C_VEL
LIN {X 0,Y 282.034,Z 638.156,A -85,B 0,C 180,E1 18557.575,E2 18557.575} C_VEL
LIN {X 0,Y 288.632,Z 654.648,A -85,B 0,C 180,E1 18563.576,E2 18563.576} C_VEL
LIN {X 0,Y 294.923,Z 676.585,A -85,B 0,C 180,E1 18569.506,E2 18569.506} C_VEL
LIN {X 0,Y 296.925,Z 688.557,A -85,B 0,C 180,E1 18572.165,E2 18572.165} C_VEL
LIN {X 0,Y 282.545,Z 725.178,A -85,B 0,C 180,E1 18575.857,E2 18575.857} C_VEL
LIN {X 0,Y 267.828,Z 755.967,A -85,B 0,C 180,E1 18580.492,E2 18580.492} C_VEL
LIN {X 0,Y 252.716,Z 783.904,A -85,B 0,C 180,E1 18586.685,E2 18586.685} C_VEL
LIN {X 0,Y 239.666,Z 806.941,A -85,B 0,C 180,E1 18594.243,E2 18594.243} C_VEL
LIN {X 0,Y 230.435,Z 824.185,A -85,B 0,C 180,E1 18602.618,E2 18602.618} C_VEL
LIN {X 0,Y 225.372,Z 836.161,A -85,B 0,C 180,E1 18611.392,E2 18611.392} C_VEL
LIN {X 0,Y 223.394,Z 843.599,A -85,B 0,C 180,E1 18620.566,E2 18620.566} C_VEL
LIN {X 0,Y 223.344,Z 846.231,A -85,B 0,C 180,E1 18630.001,E2 18630.001} C_VEL
LIN {X 0,Y 223.398,Z 843.609,A -85,B 0,C 180,E1 18639.445,E2 18639.445} C_VEL
LIN {X 0,Y 225.378,Z 836.187,A -85,B 0,C 180,E1 18648.609,E2 18648.609} C_VEL
LIN {X 0,Y 231.14,Z 822.882,A -85,B 0,C 180,E1 18658.177,E2 18658.177} C_VEL
LIN {X 0,Y 241.631,Z 803.605,A -85,B 0,C 180,E1 18667.093,E2 18667.093} C_VEL
LIN {X 0,Y 255.846,Z 778.463,A -85,B 0,C 180,E1 18674.757,E2 18674.757} C_VEL
LIN {X 0,Y 271.466,Z 748.961,A -85,B 0,C 180,E1 18680.742,E2 18680.742} C_VEL
LIN {X 0,Y 286.154,Z 717.105,A -85,B 0,C 180,E1 18685.097,E2 18685.097} C_VEL
LIN {X 0,Y 297.002,Z 687.453,A -85,B 0,C 180,E1 18688.048,E2 18688.048} C_VEL
LIN {X 0,Y 292.247,Z 665.8,A -85,B 0,C 180,E1 18693.268,E2 18693.268} C_VEL
LIN {X 0,Y 285.381,Z 645.841,A -85,B 0,C 180,E1 18699.423,E2 18699.423} C_VEL
LIN {X 0,Y 278.688,Z 630.363,A -85,B 0,C 180,E1 18706.16,E2 18706.16} C_VEL
LIN {X 0,Y 274.855,Z 623.378,A -85,B 0,C 180,E1 18711.037,E2 18711.037} C_VEL
LIN {X 0,Y 272.885,Z 618.346,A -85,B 0,C 180,E1 18715.226,E2 18715.226} C_VEL
LIN {X 0,Y 271.333,Z 616.498,A -85,B 0,C 180,E1 18721.405,E2 18721.405} C_VEL
LIN {X 0,Y 272.533,Z 618.307,A -85,B 0,C 180,E1 18728.53,E2 18728.53} C_VEL
LIN {X 0,Y 273.187,Z 622.523,A -85,B 0,C 180,E1 18731.108,E2 18731.108} C_VEL
LIN {X 0,Y 273.772,Z 633.579,A -85,B 0,C 180,E1 18735.161,E2 18735.161} C_VEL
LIN {X 0,Y 278.858,Z 645.961,A -85,B 0,C 180,E1 18741.78,E2 18741.78} C_VEL
LIN {X 0,Y 284.589,Z 663.102,A -85,B 0,C 180,E1 18748.172,E2 18748.172} C_VEL
LIN {X 0,Y 289.107,Z 683.371,A -85,B 0,C 180,E1 18753.968,E2 18753.968} C_VEL
LIN {X 0,Y 289.503,Z 691.817,A -85,B 0,C 180,E1 18755.862,E2 18755.862} C_VEL
LIN {X 0,Y 275.219,Z 723.804,A -85,B 0,C 180,E1 18759.629,E2 18759.629} C_VEL
LIN {X 0,Y 259.928,Z 751.794,A -85,B 0,C 180,E1 18764.561,E2 18764.561} C_VEL
LIN {X 0,Y 244.323,Z 776.489,A -85,B 0,C 180,E1 18771.126,E2 18771.126} C_VEL
LIN {X 0,Y 230.723,Z 796.441,A -85,B 0,C 180,E1 18779.43,E2 18779.43} C_VEL
LIN {X 0,Y 221.42,Z 810.446,A -85,B 0,C 180,E1 18788.961,E2 18788.961} C_VEL
LIN {X 0,Y 217.049,Z 818.03,A -85,B 0,C 180,E1 18797.92,E2 18797.92} C_VEL
LIN {X 0,Y 215.614,Z 821.189,A -85,B 0,C 180,E1 18805.973,E2 18805.973} C_VEL
LIN {X 0,Y 215.705,Z 821.152,A -85,B 0,C 180,E1 18814.024,E2 18814.024} C_VEL
LIN {X 0,Y 217.823,Z 816.586,A -85,B 0,C 180,E1 18824.141,E2 18824.141} C_VEL
LIN {X 0,Y 223.717,Z 806.742,A -85,B 0,C 180,E1 18833.957,E2 18833.957} C_VEL
LIN {X 0,Y 234.227,Z 791.312,A -85,B 0,C 180,E1 18842.963,E2 18842.963} C_VEL
LIN {X 0,Y 248.168,Z 770.611,A -85,B 0,C 180,E1 18850.597,E2 18850.597} C_VEL
LIN {X 0,Y 263.694,Z 745.142,A -85,B 0,C 180,E1 18856.689,E2 18856.689} C_VEL
LIN {X 0,Y 278.144,Z 717.658,A -85,B 0,C 180,E1 18861.095,E2 18861.095} C_VEL
LIN {X 0,Y 289.927,Z 690.453,A -85,B 0,C 180,E1 18864.162,E2 18864.162} C_VEL
LIN {X 0,Y 286.095,Z 668.645,A -85,B 0,C 180,E1 18869.958,E2 18869.958} C_VEL
LIN {X 0,Y 280.498,Z 650.533,A -85,B 0,C 180,E1 18876.124,E2 18876.124} C_VEL
LIN {X 0,Y 275.41,Z 637.224,A -85,B 0,C 180,E1 18882.282,E2 18882.282} C_VEL
LIN {X 0,Y 272.095,Z 630.405,A -85,B 0,C 180,E1 18887.141,E2 18887.141} C_VEL
LIN {X 0,Y 270.535,Z 625.934,A -85,B 0,C 180,E1 18891.154,E2 18891.154} C_VEL
LIN {X 0,Y 269.474,Z 623.847,A -85,B 0,C 180,E1 18900.001,E2 18900.001} C_VEL
LIN {X 0,Y 271.296,Z 627.275,A -85,B 0,C 180,E1 18906.107,E2 18906.107} C_VEL
LIN {X 0,Y 274.539,Z 635.136,A -85,B 0,C 180,E1 18911.935,E2 18911.935} C_VEL
LIN {X 0,Y 279.069,Z 645.633,A -85,B 0,C 180,E1 18917.361,E2 18917.361} C_VEL
LIN {X 0,Y 284.787,Z 661.394,A -85,B 0,C 180,E1 18923.196,E2 18923.196} C_VEL
LIN {X 0,Y 290.176,Z 683.011,A -85,B 0,C 180,E1 18929.178,E2 18929.178} C_VEL
LIN {X 0,Y 291.19,Z 692.009,A -85,B 0,C 180,E1 18931.173,E2 18931.173} C_VEL
LIN {X 0,Y 277.269,Z 725.879,A -85,B 0,C 180,E1 18934.665,E2 18934.665} C_VEL
LIN {X 0,Y 262.226,Z 756.126,A -85,B 0,C 180,E1 18939.266,E2 18939.266} C_VEL
LIN {X 0,Y 246.532,Z 783.877,A -85,B 0,C 180,E1 18945.508,E2 18945.508} C_VEL
LIN {X 0,Y 233.008,Z 806.455,A -85,B 0,C 180,E1 18953.056,E2 18953.056} C_VEL
LIN {X 0,Y 222.915,Z 824.28,A -85,B 0,C 180,E1 18961.996,E2 18961.996} C_VEL
LIN {X 0,Y 217.326,Z 836.733,A -85,B 0,C 180,E1 18971.73,E2 18971.73} C_VEL
LIN {X 0,Y 215.35,Z 843.935,A -85,B 0,C 180,E1 18981.917,E2 18981.917} C_VEL
LIN {X 0,Y 215.446,Z 845.788,A -85,B 0,C 180,E1 18990.001,E2 18990.001} C_VEL
LIN {X 0,Y 215.351,Z 843.95,A -85,B 0,C 180,E1 18998.084,E2 18998.084} C_VEL
LIN {X 0,Y 216.646,Z 838.658,A -85,B 0,C 180,E1 19006.234,E2 19006.234} C_VEL
LIN {X 0,Y 221.487,Z 827.117,A -85,B 0,C 180,E1 19016.2,E2 19016.2} C_VEL
LIN {X 0,Y 231.776,Z 808.796,A -85,B 0,C 180,E1 19026.01,E2 19026.01} C_VEL
LIN {X 0,Y 245.773,Z 785.236,A -85,B 0,C 180,E1 19034.151,E2 19034.151} C_VEL
LIN {X 0,Y 261.22,Z 758.111,A -85,B 0,C 180,E1 19040.392,E2 19040.392} C_VEL
LIN {X 0,Y 276.766,Z 727.368,A -85,B 0,C 180,E1 19045.144,E2 19045.144} C_VEL
LIN {X 0,Y 290.495,Z 694.269,A -85,B 0,C 180,E1 19048.64,E2 19048.64} C_VEL
LIN {X 0,Y 291.469,Z 690.172,A -85,B 0,C 180,E1 19049.158,E2 19049.158} C_VEL
LIN {X 0,Y 287.04,Z 669.06,A -85,B 0,C 180,E1 19054.563,E2 19054.563} C_VEL
LIN {X 0,Y 281.452,Z 651.364,A -85,B 0,C 180,E1 19060.354,E2 19060.354} C_VEL
LIN {X 0,Y 275.478,Z 636.813,A -85,B 0,C 180,E1 19067.099,E2 19067.099} C_VEL
LIN {X 0,Y 272.368,Z 630.343,A -85,B 0,C 180,E1 19071.71,E2 19071.71} C_VEL
LIN {X 0,Y 270.848,Z 625.894,A -85,B 0,C 180,E1 19075.591,E2 19075.591} C_VEL
LIN {X 0,Y 269.669,Z 624.149,A -85,B 0,C 180,E1 19079.999,E2 19079.999} C_VEL
LIN {X 0,Y 271.1,Z 626.628,A -85,B 0,C 180,E1 19089.644,E2 19089.644} C_VEL
LIN {X 0,Y 273.772,Z 633.579,A -85,B 0,C 180,E1 19095.161,E2 19095.161} C_VEL
LIN {X 0,Y 274.473,Z 642.997,A -85,B 0,C 180,E1 19098.261,E2 19098.261} C_VEL
LIN {X 0,Y 275.428,Z 652.714,A -85,B 0,C 180,E1 19101.331,E2 19101.331} C_VEL
LIN {X 0,Y 280.437,Z 669.563,A -85,B 0,C 180,E1 19107.75,E2 19107.75} C_VEL
LIN {X 0,Y 284.15,Z 690.045,A -85,B 0,C 180,E1 19113.762,E2 19113.762} C_VEL
LIN {X 0,Y 284.117,Z 694.435,A -85,B 0,C 180,E1 19114.776,E2 19114.776} C_VEL
LIN {X 0,Y 269.045,Z 726.603,A -85,B 0,C 180,E1 19118.664,E2 19118.664} C_VEL
LIN {X 0,Y 252.473,Z 755.461,A -85,B 0,C 180,E1 19123.975,E2 19123.975} C_VEL
LIN {X 0,Y 236.429,Z 779.433,A -85,B 0,C 180,E1 19130.773,E2 19130.773} C_VEL
LIN {X 0,Y 223.865,Z 796.895,A -85,B 0,C 180,E1 19138.388,E2 19138.388} C_VEL
LIN {X 0,Y 214.547,Z 810.092,A -85,B 0,C 180,E1 19147.448,E2 19147.448} C_VEL
LIN {X 0,Y 209.303,Z 818.474,A -85,B 0,C 180,E1 19157.466,E2 19157.466} C_VEL
LIN {X 0,Y 207.743,Z 821.632,A -85,B 0,C 180,E1 19165.82,E2 19165.82} C_VEL
LIN {X 0,Y 207.827,Z 821.596,A -85,B 0,C 180,E1 19174.177,E2 19174.177} C_VEL
LIN {X 0,Y 210.085,Z 817.079,A -85,B 0,C 180,E1 19184.609,E2 19184.609} C_VEL
LIN {X 0,Y 216.452,Z 807.194,A -85,B 0,C 180,E1 19194.814,E2 19194.814} C_VEL
LIN {X 0,Y 227.991,Z 791.178,A -85,B 0,C 180,E1 19204.35,E2 19204.35} C_VEL
LIN {X 0,Y 243.199,Z 769.541,A -85,B 0,C 180,E1 19212.265,E2 19212.265} C_VEL
LIN {X 0,Y 259.416,Z 743.76,A -85,B 0,C 180,E1 19218.332,E2 19218.332} C_VEL
LIN {X 0,Y 274.444,Z 715.759,A -85,B 0,C 180,E1 19222.705,E2 19222.705} C_VEL
LIN {X 0,Y 284.09,Z 694.111,A -85,B 0,C 180,E1 19225.157,E2 19225.157} C_VEL
LIN {X 0,Y 281.855,Z 676.014,A -85,B 0,C 180,E1 19230.026,E2 19230.026} C_VEL
LIN {X 0,Y 276.824,Z 657.066,A -85,B 0,C 180,E1 19236.63,E2 19236.63} C_VEL
LIN {X 0,Y 272.21,Z 643.901,A -85,B 0,C 180,E1 19242.963,E2 19242.963} C_VEL
LIN {X 0,Y 268.559,Z 633.686,A -85,B 0,C 180,E1 19250.673,E2 19250.673} C_VEL
LIN {X 0,Y 267.391,Z 631.47,A -85,B 0,C 180,E1 19260.001,E2 19260.001} C_VEL
LIN {X 0,Y 268.932,Z 634.792,A -85,B 0,C 180,E1 19265.857,E2 19265.857} C_VEL
LIN {X 0,Y 272.734,Z 644.147,A -85,B 0,C 180,E1 19272.829,E2 19272.829} C_VEL
LIN {X 0,Y 278.294,Z 659.622,A -85,B 0,C 180,E1 19279.878,E2 19279.878} C_VEL
LIN {X 0,Y 283.545,Z 679.484,A -85,B 0,C 180,E1 19286.218,E2 19286.218} C_VEL
LIN {X 0,Y 285.633,Z 695.194,A -85,B 0,C 180,E1 19290.136,E2 19290.136} C_VEL
LIN {X 0,Y 271.169,Z 728.561,A -85,B 0,C 180,E1 19293.68,E2 19293.68} C_VEL
LIN {X 0,Y 254.864,Z 759.693,A -85,B 0,C 180,E1 19298.635,E2 19298.635} C_VEL
LIN {X 0,Y 237.774,Z 788.257,A -85,B 0,C 180,E1 19305.539,E2 19305.539} C_VEL
LIN {X 0,Y 223.595,Z 810.69,A -85,B 0,C 180,E1 19313.876,E2 19313.876} C_VEL
LIN {X 0,Y 214.049,Z 826.817,A -85,B 0,C 180,E1 19322.984,E2 19322.984} C_VEL
LIN {X 0,Y 208.881,Z 838.177,A -85,B 0,C 180,E1 19333.147,E2 19333.147} C_VEL
LIN {X 0,Y 207.488,Z 843.488,A -85,B 0,C 180,E1 19341.609,E2 19341.609} C_VEL
LIN {X 0,Y 207.548,Z 845.344,A -85,B 0,C 180,E1 19350.001,E2 19350.001} C_VEL
LIN {X 0,Y 207.49,Z 843.504,A -85,B 0,C 180,E1 19358.392,E2 19358.392} C_VEL
LIN {X 0,Y 209.589,Z 836.51,A -85,B 0,C 180,E1 19368.755,E2 19368.755} C_VEL
LIN {X 0,Y 216.024,Z 823.298,A -85,B 0,C 180,E1 19379.382,E2 19379.382} C_VEL
LIN {X 0,Y 227.279,Z 804.917,A -85,B 0,C 180,E1 19388.649,E2 19388.649} C_VEL
LIN {X 0,Y 242.469,Z 780.725,A -85,B 0,C 180,E1 19396.62,E2 19396.62} C_VEL
LIN {X 0,Y 259.307,Z 751.96,A -85,B 0,C 180,E1 19402.823,E2 19402.823} C_VEL
LIN {X 0,Y 275.312,Z 720.145,A -85,B 0,C 180,E1 19407.363,E2 19407.363} C_VEL
LIN {X 0,Y 285.972,Z 693.453,A -85,B 0,C 180,E1 19410.174,E2 19410.174} C_VEL
LIN {X 0,Y 281.982,Z 672.382,A -85,B 0,C 180,E1 19415.894,E2 19415.894} C_VEL
LIN {X 0,Y 276.511,Z 653.882,A -85,B 0,C 180,E1 19422.474,E2 19422.474} C_VEL
LIN {X 0,Y 271.335,Z 640.749,A -85,B 0,C 180,E1 19429.552,E2 19429.552} C_VEL
LIN {X 0,Y 268.519,Z 633.363,A -85,B 0,C 180,E1 19435.958,E2 19435.958} C_VEL
LIN {X 0,Y 267.375,Z 631.872,A -85,B 0,C 180,E1 19443.245,E2 19443.245} C_VEL
LIN {X 0,Y 268.852,Z 634.775,A -85,B 0,C 180,E1 19449.828,E2 19449.828} C_VEL
LIN {X 0,Y 272.684,Z 644.774,A -85,B 0,C 180,E1 19457.38,E2 19457.38} C_VEL
LIN {X 0,Y 275.428,Z 652.714,A -85,B 0,C 180,E1 19461.331,E2 19461.331} C_VEL
LIN {X 0,Y 276.178,Z 660.235,A -85,B 0,C 180,E1 19463.556,E2 19463.556} C_VEL
LIN {X 0,Y 275.856,Z 674.982,A -85,B 0,C 180,E1 19467.022,E2 19467.022} C_VEL
LIN {X 0,Y 278.753,Z 694.152,A -85,B 0,C 180,E1 19472.895,E2 19472.895} C_VEL
LIN {X 0,Y 278.139,Z 698.693,A -85,B 0,C 180,E1 19473.813,E2 19473.813} C_VEL
LIN {X 0,Y 261.78,Z 731.573,A -85,B 0,C 180,E1 19477.998,E2 19477.998} C_VEL
LIN {X 0,Y 244.897,Z 759.13,A -85,B 0,C 180,E1 19483.411,E2 19483.411} C_VEL
LIN {X 0,Y 228.546,Z 782.225,A -85,B 0,C 180,E1 19490.384,E2 19490.384} C_VEL
LIN {X 0,Y 214.56,Z 800.682,A -85,B 0,C 180,E1 19499.229,E2 19499.229} C_VEL
LIN {X 0,Y 205.842,Z 812.433,A -85,B 0,C 180,E1 19508.421,E2 19508.421} C_VEL
LIN {X 0,Y 201.227,Z 819.443,A -85,B 0,C 180,E1 19517.973,E2 19517.973} C_VEL
LIN {X 0,Y 199.857,Z 822.075,A -85,B 0,C 180,E1 19525.654,E2 19525.654} C_VEL
LIN {X 0,Y 199.939,Z 822.04,A -85,B 0,C 180,E1 19534.342,E2 19534.342} C_VEL
LIN {X 0,Y 202.411,Z 817.525,A -85,B 0,C 180,E1 19545.176,E2 19545.176} C_VEL
LIN {X 0,Y 209.214,Z 807.646,A -85,B 0,C 180,E1 19555.734,E2 19555.734} C_VEL
LIN {X 0,Y 221.453,Z 791.618,A -85,B 0,C 180,E1 19565.527,E2 19565.527} C_VEL
LIN {X 0,Y 236.243,Z 771.635,A -85,B 0,C 180,E1 19573.096,E2 19573.096} C_VEL
LIN {X 0,Y 253.129,Z 746.074,A -85,B 0,C 180,E1 19579.322,E2 19579.322} C_VEL
LIN {X 0,Y 269.078,Z 717.617,A -85,B 0,C 180,E1 19583.877,E2 19583.877} C_VEL
LIN {X 0,Y 278.712,Z 696.967,A -85,B 0,C 180,E1 19586.258,E2 19586.258} C_VEL
LIN {X 0,Y 276.457,Z 678.182,A -85,B 0,C 180,E1 19591.75,E2 19591.75} C_VEL
LIN {X 0,Y 272.613,Z 662.156,A -85,B 0,C 180,E1 19597.72,E2 19597.72} C_VEL
LIN {X 0,Y 268.145,Z 648.03,A -85,B 0,C 180,E1 19605.282,E2 19605.282} C_VEL
LIN {X 0,Y 265.863,Z 641.516,A -85,B 0,C 180,E1 19611.072,E2 19611.072} C_VEL
LIN {X 0,Y 264.954,Z 639.122,A -85,B 0,C 180,E1 19616.725,E2 19616.725} C_VEL
LIN {X 0,Y 265.741,Z 640.464,A -85,B 0,C 180,E1 19623.267,E2 19623.267} C_VEL
LIN {X 0,Y 266.656,Z 643.412,A -85,B 0,C 180,E1 19626.521,E2 19626.521} C_VEL
LIN {X 0,Y 270.045,Z 652.204,A -85,B 0,C 180,E1 19632.959,E2 19632.959} C_VEL
LIN {X 0,Y 274.716,Z 667.06,A -85,B 0,C 180,E1 19639.729,E2 19639.729} C_VEL
LIN {X 0,Y 278.872,Z 685.487,A -85,B 0,C 180,E1 19645.742,E2 19645.742} C_VEL
LIN {X 0,Y 280.273,Z 698.066,A -85,B 0,C 180,E1 19649.022,E2 19649.022} C_VEL
LIN {X 0,Y 264.826,Z 731.93,A -85,B 0,C 180,E1 19652.74,E2 19652.74} C_VEL
LIN {X 0,Y 247.378,Z 763.315,A -85,B 0,C 180,E1 19658.002,E2 19658.002} C_VEL
LIN {X 0,Y 231.061,Z 789.142,A -85,B 0,C 180,E1 19664.555,E2 19664.555} C_VEL
LIN {X 0,Y 216.472,Z 811.004,A -85,B 0,C 180,E1 19672.976,E2 19672.976} C_VEL
LIN {X 0,Y 206.437,Z 826.978,A -85,B 0,C 180,E1 19682.425,E2 19682.425} C_VEL
LIN {X 0,Y 201.169,Z 837.722,A -85,B 0,C 180,E1 19692.48,E2 19692.48} C_VEL
LIN {X 0,Y 199.601,Z 843.04,A -85,B 0,C 180,E1 19701.275,E2 19701.275} C_VEL
LIN {X 0,Y 199.649,Z 844.901,A -85,B 0,C 180,E1 19710.001,E2 19710.001} C_VEL
LIN {X 0,Y 199.677,Z 842.634,A -85,B 0,C 180,E1 19719.712,E2 19719.712} C_VEL
LIN {X 0,Y 201.86,Z 836.211,A -85,B 0,C 180,E1 19729.326,E2 19729.326} C_VEL
LIN {X 0,Y 208.103,Z 824.251,A -85,B 0,C 180,E1 19739.561,E2 19739.561} C_VEL
LIN {X 0,Y 220.106,Z 805.672,A -85,B 0,C 180,E1 19749.461,E2 19749.461} C_VEL
LIN {X 0,Y 235.21,Z 782.818,A -85,B 0,C 180,E1 19757.344,E2 19757.344} C_VEL
LIN {X 0,Y 252.622,Z 754.569,A -85,B 0,C 180,E1 19763.718,E2 19763.718} C_VEL
LIN {X 0,Y 269.76,Z 722.336,A -85,B 0,C 180,E1 19768.476,E2 19768.476} C_VEL
LIN {X 0,Y 280.563,Z 697.016,A -85,B 0,C 180,E1 19771.171,E2 19771.171} C_VEL
LIN {X 0,Y 277.231,Z 676.608,A -85,B 0,C 180,E1 19777.011,E2 19777.011} C_VEL
LIN {X 0,Y 272.83,Z 660.274,A -85,B 0,C 180,E1 19783.081,E2 19783.081} C_VEL
LIN {X 0,Y 268.321,Z 647.345,A -85,B 0,C 180,E1 19790.254,E2 19790.254} C_VEL
LIN {X 0,Y 265.942,Z 640.62,A -85,B 0,C 180,E1 19796.736,E2 19796.736} C_VEL
LIN {X 0,Y 265.127,Z 639.435,A -85,B 0,C 180,E1 19803.273,E2 19803.273} C_VEL
LIN {X 0,Y 266.026,Z 641.072,A -85,B 0,C 180,E1 19808.363,E2 19808.363} C_VEL
LIN {X 0,Y 269.166,Z 650.828,A -85,B 0,C 180,E1 19816.333,E2 19816.333} C_VEL
LIN {X 0,Y 273.169,Z 663.806,A -85,B 0,C 180,E1 19822.826,E2 19822.826} C_VEL
LIN {X 0,Y 275.856,Z 674.982,A -85,B 0,C 180,E1 19827.022,E2 19827.022} C_VEL
LIN {X 0,Y 275.875,Z 683.412,A -85,B 0,C 180,E1 19829.114,E2 19829.114} C_VEL
LIN {X 0,Y 273.424,Z 699.388,A -85,B 0,C 180,E1 19832.314,E2 19832.314} C_VEL
LIN {X 0,Y 258.22,Z 729.936,A -85,B 0,C 180,E1 19836.271,E2 19836.271} C_VEL
LIN {X 0,Y 240.598,Z 758.052,A -85,B 0,C 180,E1 19841.644,E2 19841.644} C_VEL
LIN {X 0,Y 223.364,Z 781.525,A -85,B 0,C 180,E1 19848.631,E2 19848.631} C_VEL
LIN {X 0,Y 208.867,Z 799.676,A -85,B 0,C 180,E1 19857.218,E2 19857.218} C_VEL
LIN {X 0,Y 198.439,Z 812.883,A -85,B 0,C 180,E1 19867.573,E2 19867.573} C_VEL
LIN {X 0,Y 193.817,Z 819.365,A -85,B 0,C 180,E1 19876.446,E2 19876.446} C_VEL
LIN {X 0,Y 191.989,Z 822.518,A -85,B 0,C 180,E1 19885.476,E2 19885.476} C_VEL
LIN {X 0,Y 192.066,Z 822.484,A -85,B 0,C 180,E1 19894.52,E2 19894.52} C_VEL
LIN {X 0,Y 194.733,Z 817.974,A -85,B 0,C 180,E1 19905.79,E2 19905.79} C_VEL
LIN {X 0,Y 202.037,Z 808.101,A -85,B 0,C 180,E1 19916.719,E2 19916.719} C_VEL
LIN {X 0,Y 215.009,Z 792.072,A -85,B 0,C 180,E1 19926.765,E2 19926.765} C_VEL
LIN {X 0,Y 231.213,Z 771.113,A -85,B 0,C 180,E1 19934.742,E2 19934.742} C_VEL
LIN {X 0,Y 248.427,Z 745.94,A -85,B 0,C 180,E1 19940.838,E2 19940.838} C_VEL
LIN {X 0,Y 265.074,Z 717.062,A -85,B 0,C 180,E1 19945.403,E2 19945.403} C_VEL
LIN {X 0,Y 273.363,Z 699.984,A -85,B 0,C 180,E1 19947.389,E2 19947.389} C_VEL
LIN {X 0,Y 271.44,Z 681.487,A -85,B 0,C 180,E1 19953.182,E2 19953.182} C_VEL
LIN {X 0,Y 268.102,Z 666.207,A -85,B 0,C 180,E1 19959.334,E2 19959.334} C_VEL
LIN {X 0,Y 264.706,Z 653.838,A -85,B 0,C 180,E1 19966.494,E2 19966.494} C_VEL
LIN {X 0,Y 263.263,Z 648.932,A -85,B 0,C 180,E1 19971.228,E2 19971.228} C_VEL
LIN {X 0,Y 262.427,Z 646.611,A -85,B 0,C 180,E1 19976.693,E2 19976.693} C_VEL
LIN {X 0,Y 263.205,Z 647.965,A -85,B 0,C 180,E1 19983.298,E2 19983.298} C_VEL
LIN {X 0,Y 265.381,Z 654.932,A -85,B 0,C 180,E1 19989.855,E2 19989.855} C_VEL
LIN {X 0,Y 268.935,Z 666.578,A -85,B 0,C 180,E1 19996.349,E2 19996.349} C_VEL
LIN {X 0,Y 272.839,Z 683.671,A -85,B 0,C 180,E1 20002.857,E2 20002.857} C_VEL
LIN {X 0,Y 275.031,Z 700.742,A -85,B 0,C 180,E1 20007.844,E2 20007.844} C_VEL
LIN {X 0,Y 258.786,Z 734.602,A -85,B 0,C 180,E1 20011.696,E2 20011.696} C_VEL
LIN {X 0,Y 241.122,Z 764.838,A -85,B 0,C 180,E1 20016.913,E2 20016.913} C_VEL
LIN {X 0,Y 224.405,Z 790.025,A -85,B 0,C 180,E1 20023.507,E2 20023.507} C_VEL
LIN {X 0,Y 209.725,Z 810.878,A -85,B 0,C 180,E1 20031.799,E2 20031.799} C_VEL
LIN {X 0,Y 199.232,Z 826.514,A -85,B 0,C 180,E1 20041.338,E2 20041.338} C_VEL
LIN {X 0,Y 193.475,Z 837.267,A -85,B 0,C 180,E1 20051.759,E2 20051.759} C_VEL
LIN {X 0,Y 191.729,Z 842.592,A -85,B 0,C 180,E1 20060.914,E2 20060.914} C_VEL
LIN {X 0,Y 191.752,Z 844.458,A -85,B 0,C 180,E1 20070.001,E2 20070.001} C_VEL
LIN {X 0,Y 191.737,Z 842.61,A -85,B 0,C 180,E1 20079.088,E2 20079.088} C_VEL
LIN {X 0,Y 194.028,Z 836.21,A -85,B 0,C 180,E1 20089.613,E2 20089.613} C_VEL
LIN {X 0,Y 201.135,Z 823.572,A -85,B 0,C 180,E1 20100.858,E2 20100.858} C_VEL
LIN {X 0,Y 213.68,Z 805.346,A -85,B 0,C 180,E1 20110.803,E2 20110.803} C_VEL
LIN {X 0,Y 229.901,Z 782.066,A -85,B 0,C 180,E1 20118.923,E2 20118.923} C_VEL
LIN {X 0,Y 247.16,Z 755.227,A -85,B 0,C 180,E1 20125.018,E2 20125.018} C_VEL
LIN {X 0,Y 264.898,Z 723.122,A -85,B 0,C 180,E1 20129.802,E2 20129.802} C_VEL
LIN {X 0,Y 275.193,Z 699.975,A -85,B 0,C 180,E1 20132.358,E2 20132.358} C_VEL
LIN {X 0,Y 272.104,Z 679.365,A -85,B 0,C 180,E1 20138.653,E2 20138.653} C_VEL
LIN {X 0,Y 268.15,Z 663.415,A -85,B 0,C 180,E1 20145.264,E2 20145.264} C_VEL
LIN {X 0,Y 264.79,Z 653.171,A -85,B 0,C 180,E1 20151.781,E2 20151.781} C_VEL
LIN {X 0,Y 263.406,Z 648.125,A -85,B 0,C 180,E1 20156.704,E2 20156.704} C_VEL
LIN {X 0,Y 262.597,Z 646.938,A -85,B 0,C 180,E1 20163.304,E2 20163.304} C_VEL
LIN {X 0,Y 263.454,Z 648.773,A -85,B 0,C 180,E1 20168.445,E2 20168.445} C_VEL
LIN {X 0,Y 266.214,Z 658.754,A -85,B 0,C 180,E1 20176.519,E2 20176.519} C_VEL
LIN {X 0,Y 269.882,Z 673.219,A -85,B 0,C 180,E1 20183.558,E2 20183.558} C_VEL
LIN {X 0,Y 272.864,Z 691.502,A -85,B 0,C 180,E1 20189.956,E2 20189.956} C_VEL
LIN {X 0,Y 273.424,Z 699.388,A -85,B 0,C 180,E1 20192.314,E2 20192.314} C_VEL
LIN {X 0,Y 270.973,Z 706.032,A -85,B 0,C 180,E1 20193.242,E2 20193.242} C_VEL
LIN {X 0,Y 256.238,Z 726.009,A -85,B 0,C 180,E1 20194.205,E2 20194.205} C_VEL
LIN {X 0,Y 255.13,Z 727.772,A -85,B 0,C 180,E1 20194.425,E2 20194.425} C_VEL
LIN {X 0,Y 236.709,Z 756.693,A -85,B 0,C 180,E1 20199.76,E2 20199.76} C_VEL
LIN {X 0,Y 218.354,Z 780.88,A -85,B 0,C 180,E1 20206.819,E2 20206.819} C_VEL
LIN {X 0,Y 203.447,Z 798.685,A -85,B 0,C 180,E1 20215.112,E2 20215.112} C_VEL
LIN {X 0,Y 192.097,Z 812.044,A -85,B 0,C 180,E1 20225.33,E2 20225.33} C_VEL
LIN {X 0,Y 186.09,Z 819.81,A -85,B 0,C 180,E1 20235.871,E2 20235.871} C_VEL
LIN {X 0,Y 184.105,Z 822.962,A -85,B 0,C 180,E1 20245.282,E2 20245.282} C_VEL
LIN {X 0,Y 184.18,Z 822.928,A -85,B 0,C 180,E1 20254.714,E2 20254.714} C_VEL
LIN {X 0,Y 187.093,Z 818.422,A -85,B 0,C 180,E1 20266.453,E2 20266.453} C_VEL
LIN {X 0,Y 194.92,Z 808.553,A -85,B 0,C 180,E1 20277.777,E2 20277.777} C_VEL
LIN {X 0,Y 207.027,Z 794.408,A -85,B 0,C 180,E1 20287.109,E2 20287.109} C_VEL
LIN {X 0,Y 223.519,Z 774.25,A -85,B 0,C 180,E1 20295.335,E2 20295.335} C_VEL
LIN {X 0,Y 242.552,Z 747.92,A -85,B 0,C 180,E1 20302.003,E2 20302.003} C_VEL
LIN {X 0,Y 259.959,Z 718.968,A -85,B 0,C 180,E1 20306.662,E2 20306.662} C_VEL
LIN {X 0,Y 268.002,Z 702.658,A -85,B 0,C 180,E1 20308.687,E2 20308.687} C_VEL
LIN {X 0,Y 266.548,Z 685.66,A -85,B 0,C 180,E1 20314.338,E2 20314.338} C_VEL
LIN {X 0,Y 263.891,Z 670.86,A -85,B 0,C 180,E1 20320.739,E2 20320.739} C_VEL
LIN {X 0,Y 261.267,Z 660.121,A -85,B 0,C 180,E1 20327.613,E2 20327.613} C_VEL
LIN {X 0,Y 259.945,Z 655.209,A -85,B 0,C 180,E1 20333.312,E2 20333.312} C_VEL
LIN {X 0,Y 259.924,Z 653.987,A -85,B 0,C 180,E1 20340.001,E2 20340.001} C_VEL
LIN {X 0,Y 260.809,Z 656.705,A -85,B 0,C 180,E1 20344.996,E2 20344.996} C_VEL
LIN {X 0,Y 263.348,Z 666.142,A -85,B 0,C 180,E1 20352.216,E2 20352.216} C_VEL
LIN {X 0,Y 266.515,Z 679.523,A -85,B 0,C 180,E1 20358.636,E2 20358.636} C_VEL
LIN {X 0,Y 269.219,Z 697.437,A -85,B 0,C 180,E1 20364.822,E2 20364.822} C_VEL
LIN {X 0,Y 269.668,Z 703.814,A -85,B 0,C 180,E1 20366.688,E2 20366.688} C_VEL
LIN {X 0,Y 252.998,Z 736.901,A -85,B 0,C 180,E1 20370.546,E2 20370.546} C_VEL
LIN {X 0,Y 235.157,Z 766.082,A -85,B 0,C 180,E1 20375.71,E2 20375.71} C_VEL
LIN {X 0,Y 216.903,Z 792.288,A -85,B 0,C 180,E1 20382.868,E2 20382.868} C_VEL
LIN {X 0,Y 201.225,Z 813.362,A -85,B 0,C 180,E1 20391.883,E2 20391.883} C_VEL
LIN {X 0,Y 190.096,Z 829.178,A -85,B 0,C 180,E1 20402.745,E2 20402.745} C_VEL
LIN {X 0,Y 185.081,Z 838.498,A -85,B 0,C 180,E1 20413.363,E2 20413.363} C_VEL
LIN {X 0,Y 183.763,Z 842.471,A -85,B 0,C 180,E1 20421.357,E2 20421.357} C_VEL
LIN {X 0,Y 183.851,Z 844.015,A -85,B 0,C 180,E1 20430.001,E2 20430.001} C_VEL
LIN {X 0,Y 183.851,Z 842.161,A -85,B 0,C 180,E1 20439.481,E2 20439.481} C_VEL
LIN {X 0,Y 186.41,Z 835.753,A -85,B 0,C 180,E1 20450.45,E2 20450.45} C_VEL
LIN {X 0,Y 194.176,Z 823.082,A -85,B 0,C 180,E1 20462.113,E2 20462.113} C_VEL
LIN {X 0,Y 207.223,Z 805.316,A -85,B 0,C 180,E1 20472.084,E2 20472.084} C_VEL
LIN {X 0,Y 224.077,Z 782.336,A -85,B 0,C 180,E1 20480.278,E2 20480.278} C_VEL
LIN {X 0,Y 242.565,Z 754.702,A -85,B 0,C 180,E1 20486.601,E2 20486.601} C_VEL
LIN {X 0,Y 260.849,Z 722.668,A -85,B 0,C 180,E1 20491.327,E2 20491.327} C_VEL
LIN {X 0,Y 269.824,Z 703.809,A -85,B 0,C 180,E1 20493.328,E2 20493.328} C_VEL
LIN {X 0,Y 267.452,Z 683.972,A -85,B 0,C 180,E1 20499.713,E2 20499.713} C_VEL
LIN {X 0,Y 264.213,Z 669.215,A -85,B 0,C 180,E1 20506.181,E2 20506.181} C_VEL
LIN {X 0,Y 261.871,Z 660.742,A -85,B 0,C 180,E1 20511.689,E2 20511.689} C_VEL
LIN {X 0,Y 260.621,Z 655.62,A -85,B 0,C 180,E1 20516.669,E2 20516.669} C_VEL
LIN {X 0,Y 259.862,Z 654.369,A -85,B 0,C 180,E1 20523.339,E2 20523.339} C_VEL
LIN {X 0,Y 260.786,Z 657.904,A -85,B 0,C 180,E1 20530.029,E2 20530.029} C_VEL
LIN {X 0,Y 262.939,Z 666.647,A -85,B 0,C 180,E1 20536.731,E2 20536.731} C_VEL
LIN {X 0,Y 265.87,Z 680.528,A -85,B 0,C 180,E1 20543.49,E2 20543.49} C_VEL
LIN {X 0,Y 267.824,Z 697.715,A -85,B 0,C 180,E1 20549.644,E2 20549.644} C_VEL
LIN {X 0,Y 267.509,Z 704.526,A -85,B 0,C 180,E1 20551.518,E2 20551.518} C_VEL
LIN {X 0,Y 255.13,Z 727.772,A -85,B 0,C 180,E1 20554.425,E2 20554.425} C_VEL
LIN {X 0,Y 245.002,Z 740.952,A -85,B 0,C 180,E1 20555.752,E2 20555.752} C_VEL
LIN {X 0,Y 234.536,Z 753.184,A -85,B 0,C 180,E1 20557.373,E2 20557.373} C_VEL
LIN {X 0,Y 215.752,Z 777.58,A -85,B 0,C 180,E1 20564.002,E2 20564.002} C_VEL
LIN {X 0,Y 198.949,Z 796.959,A -85,B 0,C 180,E1 20572.495,E2 20572.495} C_VEL
LIN {X 0,Y 186.122,Z 811.157,A -85,B 0,C 180,E1 20582.891,E2 20582.891} C_VEL
LIN {X 0,Y 178.384,Z 820.257,A -85,B 0,C 180,E1 20595.248,E2 20595.248} C_VEL
LIN {X 0,Y 176.223,Z 823.405,A -85,B 0,C 180,E1 20605.07,E2 20605.07} C_VEL
LIN {X 0,Y 176.296,Z 823.372,A -85,B 0,C 180,E1 20614.926,E2 20614.926} C_VEL
LIN {X 0,Y 179.475,Z 818.869,A -85,B 0,C 180,E1 20627.172,E2 20627.172} C_VEL
LIN {X 0,Y 187.869,Z 809.006,A -85,B 0,C 180,E1 20638.916,E2 20638.916} C_VEL
LIN {X 0,Y 200.709,Z 794.869,A -85,B 0,C 180,E1 20648.486,E2 20648.486} C_VEL
LIN {X 0,Y 218.009,Z 774.719,A -85,B 0,C 180,E1 20656.819,E2 20656.819} C_VEL
LIN {X 0,Y 236.507,Z 750.221,A -85,B 0,C 180,E1 20663.15,E2 20663.15} C_VEL
LIN {X 0,Y 255.355,Z 720.179,A -85,B 0,C 180,E1 20668.057,E2 20668.057} C_VEL
LIN {X 0,Y 262.609,Z 705.942,A -85,B 0,C 180,E1 20669.86,E2 20669.86} C_VEL
LIN {X 0,Y 261.71,Z 689.702,A -85,B 0,C 180,E1 20675.61,E2 20675.61} C_VEL
LIN {X 0,Y 259.674,Z 675.992,A -85,B 0,C 180,E1 20681.939,E2 20681.939} C_VEL
LIN {X 0,Y 257.846,Z 666.906,A -85,B 0,C 180,E1 20688.142,E2 20688.142} C_VEL
LIN {X 0,Y 257.016,Z 662.605,A -85,B 0,C 180,E1 20693.235,E2 20693.235} C_VEL
LIN {X 0,Y 257.054,Z 661.356,A -85,B 0,C 180,E1 20700.001,E2 20700.001} C_VEL
LIN {X 0,Y 257.779,Z 664.284,A -85,B 0,C 180,E1 20705.055,E2 20705.055} C_VEL
LIN {X 0,Y 259.964,Z 673.913,A -85,B 0,C 180,E1 20712.358,E2 20712.358} C_VEL
LIN {X 0,Y 262.606,Z 687.764,A -85,B 0,C 180,E1 20718.923,E2 20718.923} C_VEL
LIN {X 0,Y 264.338,Z 706.469,A -85,B 0,C 180,E1 20725.336,E2 20725.336} C_VEL
LIN {X 0,Y 246.44,Z 740.696,A -85,B 0,C 180,E1 20729.551,E2 20729.551} C_VEL
LIN {X 0,Y 227.231,Z 770.325,A -85,B 0,C 180,E1 20735.125,E2 20735.125} C_VEL
LIN {X 0,Y 208.38,Z 795.69,A -85,B 0,C 180,E1 20742.638,E2 20742.638} C_VEL
LIN {X 0,Y 193.138,Z 814.986,A -85,B 0,C 180,E1 20751.617,E2 20751.617} C_VEL
LIN {X 0,Y 182.019,Z 829.939,A -85,B 0,C 180,E1 20762.775,E2 20762.775} C_VEL
LIN {X 0,Y 177.348,Z 838.042,A -85,B 0,C 180,E1 20772.615,E2 20772.615} C_VEL
LIN {X 0,Y 175.965,Z 841.694,A -85,B 0,C 180,E1 20780.092,E2 20780.092} C_VEL
LIN {X 0,Y 175.964,Z 843.572,A -85,B 0,C 180,E1 20790.001,E2 20790.001} C_VEL
LIN {X 0,Y 175.975,Z 841.713,A -85,B 0,C 180,E1 20799.909,E2 20799.909} C_VEL
LIN {X 0,Y 178.838,Z 835.282,A -85,B 0,C 180,E1 20811.375,E2 20811.375} C_VEL
LIN {X 0,Y 187.398,Z 822.514,A -85,B 0,C 180,E1 20823.512,E2 20823.512} C_VEL
LIN {X 0,Y 202.208,Z 803.596,A -85,B 0,C 180,E1 20834.2,E2 20834.2} C_VEL
LIN {X 0,Y 219.803,Z 780.698,A -85,B 0,C 180,E1 20842.247,E2 20842.247} C_VEL
LIN {X 0,Y 239.487,Z 752.215,A -85,B 0,C 180,E1 20848.593,E2 20848.593} C_VEL
LIN {X 0,Y 258.666,Z 718.861,A -85,B 0,C 180,E1 20853.298,E2 20853.298} C_VEL
LIN {X 0,Y 264.489,Z 706.478,A -85,B 0,C 180,E1 20854.682,E2 20854.682} C_VEL
LIN {X 0,Y 262.716,Z 687.916,A -85,B 0,C 180,E1 20861.085,E2 20861.085} C_VEL
LIN {X 0,Y 260.113,Z 674.068,A -85,B 0,C 180,E1 20867.653,E2 20867.653} C_VEL
LIN {X 0,Y 257.923,Z 664.528,A -85,B 0,C 180,E1 20874.948,E2 20874.948} C_VEL
LIN {X 0,Y 257.217,Z 661.631,A -85,B 0,C 180,E1 20879.999,E2 20879.999} C_VEL
LIN {X 0,Y 257.219,Z 662.811,A -85,B 0,C 180,E1 20886.76,E2 20886.76} C_VEL
LIN {X 0,Y 258.737,Z 670.45,A -85,B 0,C 180,E1 20894.399,E2 20894.399} C_VEL
LIN {X 0,Y 260.947,Z 682.754,A -85,B 0,C 180,E1 20901.26,E2 20901.26} C_VEL
LIN {X 0,Y 262.494,Z 698.413,A -85,B 0,C 180,E1 20907.477,E2 20907.477} C_VEL
LIN {X 0,Y 262.723,Z 706.471,A -85,B 0,C 180,E1 20910.18,E2 20910.18} C_VEL
LIN {X 0,Y 246.099,Z 735.86,A -85,B 0,C 180,E1 20914.1,E2 20914.1} C_VEL
LIN {X 0,Y 234.536,Z 753.184,A -85,B 0,C 180,E1 20917.373,E2 20917.373} C_VEL
LIN {X 0,Y 223.69,Z 764.728,A -85,B 0,C 180,E1 20919.273,E2 20919.273} C_VEL
LIN {X 0,Y 212.649,Z 775.298,A -85,B 0,C 180,E1 20921.515,E2 20921.515} C_VEL
LIN {X 0,Y 194.414,Z 795.536,A -85,B 0,C 180,E1 20930.021,E2 20930.021} C_VEL
LIN {X 0,Y 180.862,Z 809.601,A -85,B 0,C 180,E1 20939.848,E2 20939.848} C_VEL
LIN {X 0,Y 171.83,Z 819.407,A -85,B 0,C 180,E1 20952.036,E2 20952.036} C_VEL
LIN {X 0,Y 168.343,Z 823.849,A -85,B 0,C 180,E1 20964.839,E2 20964.839} C_VEL
LIN {X 0,Y 168.415,Z 823.816,A -85,B 0,C 180,E1 20975.157,E2 20975.157} C_VEL
LIN {X 0,Y 171.892,Z 819.317,A -85,B 0,C 180,E1 20987.955,E2 20987.955} C_VEL
LIN {X 0,Y 180.908,Z 809.46,A -85,B 0,C 180,E1 21000.141,E2 21000.141} C_VEL
LIN {X 0,Y 196.298,Z 793.449,A -85,B 0,C 180,E1 21010.965,E2 21010.965} C_VEL
LIN {X 0,Y 214.906,Z 772.553,A -85,B 0,C 180,E1 21019.23,E2 21019.23} C_VEL
LIN {X 0,Y 234.385,Z 747.06,A -85,B 0,C 180,E1 21025.446,E2 21025.446} C_VEL
LIN {X 0,Y 252.65,Z 718.247,A -85,B 0,C 180,E1 21029.903,E2 21029.903} C_VEL
LIN {X 0,Y 257.172,Z 710.006,A -85,B 0,C 180,E1 21030.885,E2 21030.885} C_VEL
LIN {X 0,Y 257.029,Z 695.497,A -85,B 0,C 180,E1 21036.193,E2 21036.193} C_VEL
LIN {X 0,Y 255.617,Z 681.907,A -85,B 0,C 180,E1 21042.775,E2 21042.775} C_VEL
LIN {X 0,Y 254.242,Z 672.563,A -85,B 0,C 180,E1 21049.71,E2 21049.71} C_VEL
LIN {X 0,Y 253.645,Z 668.685,A -85,B 0,C 180,E1 21056.579,E2 21056.579} C_VEL
LIN {X 0,Y 253.883,Z 668.605,A -85,B 0,C 180,E1 21060.001,E2 21060.001} C_VEL
LIN {X 0,Y 254.497,Z 671.729,A -85,B 0,C 180,E1 21065.12,E2 21065.12} C_VEL
LIN {X 0,Y 256.124,Z 680.552,A -85,B 0,C 180,E1 21071.94,E2 21071.94} C_VEL
LIN {X 0,Y 258.195,Z 694.841,A -85,B 0,C 180,E1 21078.816,E2 21078.816} C_VEL
LIN {X 0,Y 259.137,Z 709.856,A -85,B 0,C 180,E1 21084.14,E2 21084.14} C_VEL
LIN {X 0,Y 240.078,Z 744.05,A -85,B 0,C 180,E1 21088.483,E2 21088.483} C_VEL
LIN {X 0,Y 221.299,Z 771.577,A -85,B 0,C 180,E1 21093.829,E2 21093.829} C_VEL
LIN {X 0,Y 201.867,Z 796.454,A -85,B 0,C 180,E1 21101.409,E2 21101.409} C_VEL
LIN {X 0,Y 185.517,Z 816.02,A -85,B 0,C 180,E1 21110.981,E2 21110.981} C_VEL
LIN {X 0,Y 173.925,Z 830.699,A -85,B 0,C 180,E1 21122.806,E2 21122.806} C_VEL
LIN {X 0,Y 168.93,Z 839.004,A -85,B 0,C 180,E1 21134.404,E2 21134.404} C_VEL
LIN {X 0,Y 167.777,Z 842.618,A -85,B 0,C 180,E1 21144.823,E2 21144.823} C_VEL
LIN {X 0,Y 168.061,Z 843.129,A -85,B 0,C 180,E1 21150.001,E2 21150.001} C_VEL
LIN {X 0,Y 168.109,Z 841.265,A -85,B 0,C 180,E1 21160.378,E2 21160.378} C_VEL
LIN {X 0,Y 171.275,Z 834.822,A -85,B 0,C 180,E1 21172.369,E2 21172.369} C_VEL
LIN {X 0,Y 180.075,Z 822.75,A -85,B 0,C 180,E1 21184.433,E2 21184.433} C_VEL
LIN {X 0,Y 195.634,Z 804.025,A -85,B 0,C 180,E1 21195.466,E2 21195.466} C_VEL
LIN {X 0,Y 214.223,Z 781.075,A -85,B 0,C 180,E1 21203.724,E2 21203.724} C_VEL
LIN {X 0,Y 234.002,Z 753.662,A -85,B 0,C 180,E1 21209.929,E2 21209.929} C_VEL
LIN {X 0,Y 253.849,Z 720.762,A -85,B 0,C 180,E1 21214.648,E2 21214.648} C_VEL
LIN {X 0,Y 259.285,Z 709.889,A -85,B 0,C 180,E1 21215.875,E2 21215.875} C_VEL
LIN {X 0,Y 258.066,Z 692.934,A -85,B 0,C 180,E1 21222.037,E2 21222.037} C_VEL
LIN {X 0,Y 256.265,Z 680.718,A -85,B 0,C 180,E1 21228.066,E2 21228.066} C_VEL
LIN {X 0,Y 254.634,Z 671.988,A -85,B 0,C 180,E1 21234.883,E2 21234.883} C_VEL
LIN {X 0,Y 254.037,Z 668.869,A -85,B 0,C 180,E1 21239.999,E2 21239.999} C_VEL
LIN {X 0,Y 254.009,Z 670.123,A -85,B 0,C 180,E1 21246.846,E2 21246.846} C_VEL
LIN {X 0,Y 254.967,Z 676.837,A -85,B 0,C 180,E1 21253.739,E2 21253.739} C_VEL
LIN {X 0,Y 256.573,Z 688.883,A -85,B 0,C 180,E1 21260.734,E2 21260.734} C_VEL
LIN {X 0,Y 257.461,Z 704.759,A -85,B 0,C 180,E1 21267.195,E2 21267.195} C_VEL
LIN {X 0,Y 257.139,Z 710.459,A -85,B 0,C 180,E1 21269.068,E2 21269.068} C_VEL
LIN {X 0,Y 237.943,Z 742.203,A -85,B 0,C 180,E1 21273.541,E2 21273.541} C_VEL
LIN {X 0,Y 218.003,Z 768.869,A -85,B 0,C 180,E1 21279.559,E2 21279.559} C_VEL
LIN {X 0,Y 212.649,Z 775.298,A -85,B 0,C 180,E1 21281.515,E2 21281.515} C_VEL
LIN {X 0,Y 201.511,Z 785.024,A -85,B 0,C 180,E1 21284.153,E2 21284.153} C_VEL
LIN {X 0,Y 190.598,Z 793.732,A -85,B 0,C 180,E1 21287.23,E2 21287.23} C_VEL
LIN {X 0,Y 175.291,Z 808.777,A -85,B 0,C 180,E1 21297.326,E2 21297.326} C_VEL
LIN {X 0,Y 165.724,Z 818.379,A -85,B 0,C 180,E1 21308.564,E2 21308.564} C_VEL
LIN {X 0,Y 161.327,Z 823.11,A -85,B 0,C 180,E1 21319.18,E2 21319.18} C_VEL
LIN {X 0,Y 160.46,Z 824.692,A -85,B 0,C 180,E1 21329.999,E2 21329.999} C_VEL
LIN {X 0,Y 161.369,Z 823.06,A -85,B 0,C 180,E1 21340.815,E2 21340.815} C_VEL
LIN {X 0,Y 167.456,Z 816.5,A -85,B 0,C 180,E1 21354.007,E2 21354.007} C_VEL
LIN {X 0,Y 179.815,Z 804.326,A -85,B 0,C 180,E1 21366.114,E2 21366.114} C_VEL
LIN {X 0,Y 196.911,Z 787.147,A -85,B 0,C 180,E1 21375.758,E2 21375.758} C_VEL
LIN {X 0,Y 217.607,Z 763.648,A -85,B 0,C 180,E1 21383.512,E2 21383.512} C_VEL
LIN {X 0,Y 237.182,Z 737.244,A -85,B 0,C 180,E1 21388.89,E2 21388.89} C_VEL
LIN {X 0,Y 252.143,Z 712.587,A -85,B 0,C 180,E1 21392.34,E2 21392.34} C_VEL
LIN {X 0,Y 252.09,Z 696.518,A -85,B 0,C 180,E1 21398.88,E2 21398.88} C_VEL
LIN {X 0,Y 251.208,Z 685.461,A -85,B 0,C 180,E1 21405.072,E2 21405.072} C_VEL
LIN {X 0,Y 250.548,Z 678.232,A -85,B 0,C 180,E1 21411.312,E2 21411.312} C_VEL
LIN {X 0,Y 250.31,Z 675.893,A -85,B 0,C 180,E1 21416.533,E2 21416.533} C_VEL
LIN {X 0,Y 250.572,Z 675.806,A -85,B 0,C 180,E1 21420.001,E2 21420.001} C_VEL
LIN {X 0,Y 251.004,Z 679.048,A -85,B 0,C 180,E1 21425.191,E2 21425.191} C_VEL
LIN {X 0,Y 252.364,Z 688.396,A -85,B 0,C 180,E1 21432.276,E2 21432.276} C_VEL
LIN {X 0,Y 253.597,Z 701.295,A -85,B 0,C 180,E1 21438.492,E2 21438.492} C_VEL
LIN {X 0,Y 253.857,Z 713.022,A -85,B 0,C 180,E1 21442.834,E2 21442.834} C_VEL
LIN {X 0,Y 235.195,Z 745.188,A -85,B 0,C 180,E1 21447.011,E2 21447.011} C_VEL
LIN {X 0,Y 215.393,Z 772.944,A -85,B 0,C 180,E1 21452.489,E2 21452.489} C_VEL
LIN {X 0,Y 195.285,Z 797.411,A -85,B 0,C 180,E1 21460.174,E2 21460.174} C_VEL
LIN {X 0,Y 177.725,Z 817.267,A -85,B 0,C 180,E1 21470.423,E2 21470.423} C_VEL
LIN {X 0,Y 165.825,Z 831.449,A -85,B 0,C 180,E1 21482.838,E2 21482.838} C_VEL
LIN {X 0,Y 160.614,Z 839.845,A -85,B 0,C 180,E1 21496.37,E2 21496.37} C_VEL
LIN {X 0,Y 159.876,Z 842.172,A -85,B 0,C 180,E1 21504.567,E2 21504.567} C_VEL
LIN {X 0,Y 160.165,Z 842.685,A -85,B 0,C 180,E1 21510.001,E2 21510.001} C_VEL
LIN {X 0,Y 160.249,Z 840.816,A -85,B 0,C 180,E1 21520.893,E2 21520.893} C_VEL
LIN {X 0,Y 163.062,Z 835.48,A -85,B 0,C 180,E1 21531.803,E2 21531.803} C_VEL
LIN {X 0,Y 172.192,Z 823.647,A -85,B 0,C 180,E1 21544.858,E2 21544.858} C_VEL
LIN {X 0,Y 188.325,Z 805.454,A -85,B 0,C 180,E1 21556.351,E2 21556.351} C_VEL
LIN {X 0,Y 207.971,Z 782.468,A -85,B 0,C 180,E1 21564.987,E2 21564.987} C_VEL
LIN {X 0,Y 228.643,Z 755.108,A -85,B 0,C 180,E1 21571.332,E2 21571.332} C_VEL
LIN {X 0,Y 247.956,Z 724.619,A -85,B 0,C 180,E1 21575.799,E2 21575.799} C_VEL
LIN {X 0,Y 253.997,Z 713.117,A -85,B 0,C 180,E1 21577.166,E2 21577.166} C_VEL
LIN {X 0,Y 253.414,Z 697.018,A -85,B 0,C 180,E1 21583.424,E2 21583.424} C_VEL
LIN {X 0,Y 252.123,Z 685.527,A -85,B 0,C 180,E1 21589.621,E2 21589.621} C_VEL
LIN {X 0,Y 251.023,Z 677.697,A -85,B 0,C 180,E1 21596.542,E2 21596.542} C_VEL
LIN {X 0,Y 250.711,Z 676.071,A -85,B 0,C 180,E1 21599.999,E2 21599.999} C_VEL
LIN {X 0,Y 250.577,Z 677.357,A -85,B 0,C 180,E1 21606.94,E2 21606.94} C_VEL
LIN {X 0,Y 251.268,Z 684.341,A -85,B 0,C 180,E1 21613.945,E2 21613.945} C_VEL
LIN {X 0,Y 252.136,Z 694.996,A -85,B 0,C 180,E1 21620.208,E2 21620.208} C_VEL
LIN {X 0,Y 252.278,Z 710.511,A -85,B 0,C 180,E1 21626.746,E2 21626.746} C_VEL
LIN {X 0,Y 251.677,Z 714.165,A -85,B 0,C 180,E1 21627.86,E2 21627.86} C_VEL
LIN {X 0,Y 232.577,Z 744.191,A -85,B 0,C 180,E1 21632.189,E2 21632.189} C_VEL
LIN {X 0,Y 213.706,Z 768.544,A -85,B 0,C 180,E1 21637.679,E2 21637.679} C_VEL
LIN {X 0,Y 194.173,Z 790.041,A -85,B 0,C 180,E1 21645.43,E2 21645.43} C_VEL
LIN {X 0,Y 190.598,Z 793.732,A -85,B 0,C 180,E1 21647.23,E2 21647.23} C_VEL
LIN {X 0,Y 179.978,Z 801.514,A -85,B 0,C 180,E1 21650.816,E2 21650.816} C_VEL
LIN {X 0,Y 169.771,Z 808.209,A -85,B 0,C 180,E1 21654.949,E2 21654.949} C_VEL
LIN {X 0,Y 158.328,Z 818.825,A -85,B 0,C 180,E1 21667.51,E2 21667.51} C_VEL
LIN {X 0,Y 152.789,Z 824.395,A -85,B 0,C 180,E1 21682.245,E2 21682.245} C_VEL
LIN {X 0,Y 152.566,Z 825.135,A -85,B 0,C 180,E1 21689.999,E2 21689.999} C_VEL
LIN {X 0,Y 153.582,Z 823.505,A -85,B 0,C 180,E1 21701.37,E2 21701.37} C_VEL
LIN {X 0,Y 160.079,Z 817.063,A -85,B 0,C 180,E1 21714.999,E2 21714.999} C_VEL
LIN {X 0,Y 173.428,Z 804.778,A -85,B 0,C 180,E1 21727.669,E2 21727.669} C_VEL
LIN {X 0,Y 192.15,Z 786.882,A -85,B 0,C 180,E1 21737.775,E2 21737.775} C_VEL
LIN {X 0,Y 212.65,Z 764.515,A -85,B 0,C 180,E1 21745.142,E2 21745.142} C_VEL
LIN {X 0,Y 233.368,Z 737.505,A -85,B 0,C 180,E1 21750.599,E2 21750.599} C_VEL
LIN {X 0,Y 246.938,Z 715.968,A -85,B 0,C 180,E1 21753.61,E2 21753.61} C_VEL
LIN {X 0,Y 247.43,Z 700.61,A -85,B 0,C 180,E1 21760.335,E2 21760.335} C_VEL
LIN {X 0,Y 247.046,Z 690.126,A -85,B 0,C 180,E1 21766.805,E2 21766.805} C_VEL
LIN {X 0,Y 246.841,Z 684.288,A -85,B 0,C 180,E1 21772.955,E2 21772.955} C_VEL
LIN {X 0,Y 247.034,Z 682.916,A -85,B 0,C 180,E1 21780.001,E2 21780.001} C_VEL
LIN {X 0,Y 247.355,Z 686.327,A -85,B 0,C 180,E1 21785.278,E2 21785.278} C_VEL
LIN {X 0,Y 248.151,Z 694.427,A -85,B 0,C 180,E1 21791.613,E2 21791.613} C_VEL
LIN {X 0,Y 248.837,Z 707.684,A -85,B 0,C 180,E1 21798.169,E2 21798.169} C_VEL
LIN {X 0,Y 248.565,Z 716.973,A -85,B 0,C 180,E1 21801.704,E2 21801.704} C_VEL
LIN {X 0,Y 228.638,Z 749.103,A -85,B 0,C 180,E1 21805.93,E2 21805.93} C_VEL
LIN {X 0,Y 207.175,Z 777.323,A -85,B 0,C 180,E1 21811.837,E2 21811.837} C_VEL
LIN {X 0,Y 186.291,Z 801.074,A -85,B 0,C 180,E1 21820.03,E2 21820.03} C_VEL
LIN {X 0,Y 168.428,Z 819.973,A -85,B 0,C 180,E1 21831.006,E2 21831.006} C_VEL
LIN {X 0,Y 156.953,Z 833.063,A -85,B 0,C 180,E1 21844.274,E2 21844.274} C_VEL
LIN {X 0,Y 152.831,Z 839.395,A -85,B 0,C 180,E1 21855.662,E2 21855.662} C_VEL
LIN {X 0,Y 151.961,Z 841.878,A -85,B 0,C 180,E1 21865.063,E2 21865.063} C_VEL
LIN {X 0,Y 152.26,Z 842.242,A -85,B 0,C 180,E1 21870.001,E2 21870.001} C_VEL
LIN {X 0,Y 152.425,Z 840.369,A -85,B 0,C 180,E1 21881.46,E2 21881.46} C_VEL
LIN {X 0,Y 155.533,Z 835.024,A -85,B 0,C 180,E1 21892.917,E2 21892.917} C_VEL
LIN {X 0,Y 165.541,Z 823.186,A -85,B 0,C 180,E1 21906.478,E2 21906.478} C_VEL
LIN {X 0,Y 182.755,Z 804.978,A -85,B 0,C 180,E1 21918.213,E2 21918.213} C_VEL
LIN {X 0,Y 203.35,Z 781.973,A -85,B 0,C 180,E1 21926.891,E2 21926.891} C_VEL
LIN {X 0,Y 224.681,Z 754.828,A -85,B 0,C 180,E1 21933.109,E2 21933.109} C_VEL
LIN {X 0,Y 244.749,Z 724.045,A -85,B 0,C 180,E1 21937.528,E2 21937.528} C_VEL
LIN {X 0,Y 248.8,Z 716.178,A -85,B 0,C 180,E1 21938.586,E2 21938.586} C_VEL
LIN {X 0,Y 248.726,Z 701.31,A -85,B 0,C 180,E1 21944.758,E2 21944.758} C_VEL
LIN {X 0,Y 247.853,Z 690.467,A -85,B 0,C 180,E1 21951.216,E2 21951.216} C_VEL
LIN {X 0,Y 247.431,Z 684.922,A -85,B 0,C 180,E1 21956.491,E2 21956.491} C_VEL
LIN {X 0,Y 247.172,Z 683.178,A -85,B 0,C 180,E1 21959.999,E2 21959.999} C_VEL
LIN {X 0,Y 246.99,Z 684.548,A -85,B 0,C 180,E1 21967.041,E2 21967.041} C_VEL
LIN {X 0,Y 247.247,Z 691.801,A -85,B 0,C 180,E1 21974.177,E2 21974.177} C_VEL
LIN {X 0,Y 247.606,Z 702.808,A -85,B 0,C 180,E1 21980.583,E2 21980.583} C_VEL
LIN {X 0,Y 246.971,Z 716.081,A -85,B 0,C 180,E1 21986.246,E2 21986.246} C_VEL
LIN {X 0,Y 228.442,Z 744.693,A -85,B 0,C 180,E1 21990.502,E2 21990.502} C_VEL
LIN {X 0,Y 208.682,Z 769.286,A -85,B 0,C 180,E1 21996.022,E2 21996.022} C_VEL
LIN {X 0,Y 188.564,Z 790.5,A -85,B 0,C 180,E1 22003.726,E2 22003.726} C_VEL
LIN {X 0,Y 170.143,Z 807.885,A -85,B 0,C 180,E1 22014.66,E2 22014.66} C_VEL
LIN {X 0,Y 169.771,Z 808.209,A -85,B 0,C 180,E1 22014.949,E2 22014.949} C_VEL
LIN {X 0,Y 160.326,Z 813.861,A -85,B 0,C 180,E1 22019.701,E2 22019.701} C_VEL
LIN {X 0,Y 151.838,Z 818.482,A -85,B 0,C 180,E1 22025.083,E2 22025.083} C_VEL
LIN {X 0,Y 145.774,Z 824,A -85,B 0,C 180,E1 22038.01,E2 22038.01} C_VEL
LIN {X 0,Y 144.691,Z 825.577,A -85,B 0,C 180,E1 22049.999,E2 22049.999} C_VEL
LIN {X 0,Y 145.81,Z 823.951,A -85,B 0,C 180,E1 22061.985,E2 22061.985} C_VEL
LIN {X 0,Y 152.505,Z 817.837,A -85,B 0,C 180,E1 22075.773,E2 22075.773} C_VEL
LIN {X 0,Y 165.417,Z 806.705,A -85,B 0,C 180,E1 22088.156,E2 22088.156} C_VEL
LIN {X 0,Y 184.582,Z 789.484,A -85,B 0,C 180,E1 22098.63,E2 22098.63} C_VEL
LIN {X 0,Y 206.814,Z 766.643,A -85,B 0,C 180,E1 22106.524,E2 22106.524} C_VEL
LIN {X 0,Y 228.172,Z 740.014,A -85,B 0,C 180,E1 22112.014,E2 22112.014} C_VEL
LIN {X 0,Y 241.848,Z 719.134,A -85,B 0,C 180,E1 22115.027,E2 22115.027} C_VEL
LIN {X 0,Y 242.855,Z 704.77,A -85,B 0,C 180,E1 22121.839,E2 22121.839} C_VEL
LIN {X 0,Y 242.945,Z 694.963,A -85,B 0,C 180,E1 22128.656,E2 22128.656} C_VEL
LIN {X 0,Y 242.982,Z 691.291,A -85,B 0,C 180,E1 22132.842,E2 22132.842} C_VEL
LIN {X 0,Y 243.261,Z 689.91,A -85,B 0,C 180,E1 22140.001,E2 22140.001} C_VEL
LIN {X 0,Y 243.437,Z 693.747,A -85,B 0,C 180,E1 22145.672,E2 22145.672} C_VEL
LIN {X 0,Y 243.853,Z 701.849,A -85,B 0,C 180,E1 22151.821,E2 22151.821} C_VEL
LIN {X 0,Y 243.855,Z 714.486,A -85,B 0,C 180,E1 22158.085,E2 22158.085} C_VEL
LIN {X 0,Y 243.279,Z 720.629,A -85,B 0,C 180,E1 22160.381,E2 22160.381} C_VEL
LIN {X 0,Y 222.912,Z 751.709,A -85,B 0,C 180,E1 22164.589,E2 22164.589} C_VEL
LIN {X 0,Y 200.311,Z 779.836,A -85,B 0,C 180,E1 22170.71,E2 22170.71} C_VEL
LIN {X 0,Y 180.216,Z 801.493,A -85,B 0,C 180,E1 22178.448,E2 22178.448} C_VEL
LIN {X 0,Y 162.137,Z 819.506,A -85,B 0,C 180,E1 22189.183,E2 22189.183} C_VEL
LIN {X 0,Y 149.647,Z 832.603,A -85,B 0,C 180,E1 22202.918,E2 22202.918} C_VEL
LIN {X 0,Y 145.084,Z 838.945,A -85,B 0,C 180,E1 22214.878,E2 22214.878} C_VEL
LIN {X 0,Y 144.077,Z 841.28,A -85,B 0,C 180,E1 22223.969,E2 22223.969} C_VEL
LIN {X 0,Y 144.364,Z 841.799,A -85,B 0,C 180,E1 22230.001,E2 22230.001} C_VEL
LIN {X 0,Y 144.584,Z 839.919,A -85,B 0,C 180,E1 22242.09,E2 22242.09} C_VEL
LIN {X 0,Y 148.072,Z 834.567,A -85,B 0,C 180,E1 22254.144,E2 22254.144} C_VEL
LIN {X 0,Y 159.03,Z 822.725,A -85,B 0,C 180,E1 22268.232,E2 22268.232} C_VEL
LIN {X 0,Y 177.393,Z 804.504,A -85,B 0,C 180,E1 22280.19,E2 22280.19} C_VEL
LIN {X 0,Y 199.002,Z 781.485,A -85,B 0,C 180,E1 22288.863,E2 22288.863} C_VEL
LIN {X 0,Y 220.675,Z 754.887,A -85,B 0,C 180,E1 22294.894,E2 22294.894} C_VEL
LIN {X 0,Y 241.755,Z 723.472,A -85,B 0,C 180,E1 22299.311,E2 22299.311} C_VEL
LIN {X 0,Y 243.681,Z 719.932,A -85,B 0,C 180,E1 22299.822,E2 22299.822} C_VEL
LIN {X 0,Y 244.097,Z 705.386,A -85,B 0,C 180,E1 22306.262,E2 22306.262} C_VEL
LIN {X 0,Y 243.65,Z 695.577,A -85,B 0,C 180,E1 22312.861,E2 22312.861} C_VEL
LIN {X 0,Y 243.519,Z 692.018,A -85,B 0,C 180,E1 22316.435,E2 22316.435} C_VEL
LIN {X 0,Y 243.394,Z 690.152,A -85,B 0,C 180,E1 22319.999,E2 22319.999} C_VEL
LIN {X 0,Y 243.107,Z 691.59,A -85,B 0,C 180,E1 22327.154,E2 22327.154} C_VEL
LIN {X 0,Y 243.004,Z 699.115,A -85,B 0,C 180,E1 22334.43,E2 22334.43} C_VEL
LIN {X 0,Y 242.67,Z 710.644,A -85,B 0,C 180,E1 22341.021,E2 22341.021} C_VEL
LIN {X 0,Y 241.827,Z 719.634,A -85,B 0,C 180,E1 22344.972,E2 22344.972} C_VEL
LIN {X 0,Y 221.68,Z 748.956,A -85,B 0,C 180,E1 22349.446,E2 22349.446} C_VEL
LIN {X 0,Y 198.71,Z 775.576,A -85,B 0,C 180,E1 22355.946,E2 22355.946} C_VEL
LIN {X 0,Y 178.763,Z 795.021,A -85,B 0,C 180,E1 22363.951,E2 22363.951} C_VEL
LIN {X 0,Y 162.089,Z 809.673,A -85,B 0,C 180,E1 22374.28,E2 22374.28} C_VEL
LIN {X 0,Y 151.838,Z 818.482,A -85,B 0,C 180,E1 22385.083,E2 22385.083} C_VEL
LIN {X 0,Y 146.581,Z 821.298,A -85,B 0,C 180,E1 22389.568,E2 22389.568} C_VEL
LIN {X 0,Y 138.304,Z 824.312,A -85,B 0,C 180,E1 22396.732,E2 22396.732} C_VEL
LIN {X 0,Y 137.937,Z 824.501,A -85,B 0,C 180,E1 22397.629,E2 22397.629} C_VEL
LIN {X 0,Y 136.796,Z 826.02,A -85,B 0,C 180,E1 22409.999,E2 22409.999} C_VEL
LIN {X 0,Y 138.062,Z 824.397,A -85,B 0,C 180,E1 22422.668,E2 22422.668} C_VEL
LIN {X 0,Y 145.093,Z 818.497,A -85,B 0,C 180,E1 22436.806,E2 22436.806} C_VEL
LIN {X 0,Y 159.21,Z 807.159,A -85,B 0,C 180,E1 22449.933,E2 22449.933} C_VEL
LIN {X 0,Y 177.99,Z 791.203,A -85,B 0,C 180,E1 22459.957,E2 22459.957} C_VEL
LIN {X 0,Y 199.945,Z 769.821,A -85,B 0,C 180,E1 22467.667,E2 22467.667} C_VEL
LIN {X 0,Y 222.363,Z 743.489,A -85,B 0,C 180,E1 22473.313,E2 22473.313} C_VEL
LIN {X 0,Y 236.136,Z 724.079,A -85,B 0,C 180,E1 22476.066,E2 22476.066} C_VEL
LIN {X 0,Y 237.866,Z 713.511,A -85,B 0,C 180,E1 22480.833,E2 22480.833} C_VEL
LIN {X 0,Y 238.583,Z 703.596,A -85,B 0,C 180,E1 22487.169,E2 22487.169} C_VEL
LIN {X 0,Y 238.934,Z 698.267,A -85,B 0,C 180,E1 22492.72,E2 22492.72} C_VEL
LIN {X 0,Y 239.359,Z 696.827,A -85,B 0,C 180,E1 22500.001,E2 22500.001} C_VEL
LIN {X 0,Y 239.3,Z 700.778,A -85,B 0,C 180,E1 22505.771,E2 22505.771} C_VEL
LIN {X 0,Y 239.341,Z 708.946,A -85,B 0,C 180,E1 22511.864,E2 22511.864} C_VEL
LIN {X 0,Y 238.704,Z 721.093,A -85,B 0,C 180,E1 22517.935,E2 22517.935} C_VEL
LIN {X 0,Y 238.109,Z 724.034,A -85,B 0,C 180,E1 22519.01,E2 22519.01} C_VEL
LIN {X 0,Y 217.046,Z 754.569,A -85,B 0,C 180,E1 22523.238,E2 22523.238} C_VEL
LIN {X 0,Y 194.881,Z 780.846,A -85,B 0,C 180,E1 22529.072,E2 22529.072} C_VEL
LIN {X 0,Y 172.259,Z 803.926,A -85,B 0,C 180,E1 22537.718,E2 22537.718} C_VEL
LIN {X 0,Y 152.654,Z 822.199,A -85,B 0,C 180,E1 22549.86,E2 22549.86} C_VEL
LIN {X 0,Y 140.684,Z 834.074,A -85,B 0,C 180,E1 22564.503,E2 22564.503} C_VEL
LIN {X 0,Y 136.75,Z 839.447,A -85,B 0,C 180,E1 22577.208,E2 22577.208} C_VEL
LIN {X 0,Y 136.485,Z 841.357,A -85,B 0,C 180,E1 22590.001,E2 22590.001} C_VEL
LIN {X 0,Y 136.762,Z 839.47,A -85,B 0,C 180,E1 22602.793,E2 22602.793} C_VEL
LIN {X 0,Y 142.419,Z 832.187,A -85,B 0,C 180,E1 22618.582,E2 22618.582} C_VEL
LIN {X 0,Y 156.027,Z 819.114,A -85,B 0,C 180,E1 22632.788,E2 22632.788} C_VEL
LIN {X 0,Y 175.735,Z 800.647,A -85,B 0,C 180,E1 22643.874,E2 22643.874} C_VEL
LIN {X 0,Y 199.057,Z 776.488,A -85,B 0,C 180,E1 22652.156,E2 22652.156} C_VEL
LIN {X 0,Y 222.437,Z 747.651,A -85,B 0,C 180,E1 22657.936,E2 22657.936} C_VEL
LIN {X 0,Y 238.186,Z 724.246,A -85,B 0,C 180,E1 22660.977,E2 22660.977} C_VEL
LIN {X 0,Y 239.297,Z 714.121,A -85,B 0,C 180,E1 22665.34,E2 22665.34} C_VEL
LIN {X 0,Y 239.479,Z 703.649,A -85,B 0,C 180,E1 22671.822,E2 22671.822} C_VEL
LIN {X 0,Y 239.467,Z 699.031,A -85,B 0,C 180,E1 22676.375,E2 22676.375} C_VEL
LIN {X 0,Y 239.476,Z 697.071,A -85,B 0,C 180,E1 22679.999,E2 22679.999} C_VEL
LIN {X 0,Y 239.03,Z 698.583,A -85,B 0,C 180,E1 22687.277,E2 22687.277} C_VEL
LIN {X 0,Y 238.644,Z 705.114,A -85,B 0,C 180,E1 22693.762,E2 22693.762} C_VEL
LIN {X 0,Y 237.692,Z 716.35,A -85,B 0,C 180,E1 22700.475,E2 22700.475} C_VEL
LIN {X 0,Y 236.085,Z 724.437,A -85,B 0,C 180,E1 22703.864,E2 22703.864} C_VEL
LIN {X 0,Y 214.982,Z 753.028,A -85,B 0,C 180,E1 22708.316,E2 22708.316} C_VEL
LIN {X 0,Y 192.814,Z 777.336,A -85,B 0,C 180,E1 22714.461,E2 22714.461} C_VEL
LIN {X 0,Y 171.117,Z 797.36,A -85,B 0,C 180,E1 22723.115,E2 22723.115} C_VEL
LIN {X 0,Y 152.461,Z 812.683,A -85,B 0,C 180,E1 22735.177,E2 22735.177} C_VEL
LIN {X 0,Y 141.883,Z 821.192,A -85,B 0,C 180,E1 22748.068,E2 22748.068} C_VEL
LIN {X 0,Y 137.937,Z 824.501,A -85,B 0,C 180,E1 22757.629,E2 22757.629} C_VEL
LIN {X 0,Y 132.896,Z 826.005,A -85,B 0,C 180,E1 22764.679,E2 22764.679} C_VEL
LIN {X 0,Y 128.782,Z 826.323,A -85,B 0,C 180,E1 22772.204,E2 22772.204} C_VEL
LIN {X 0,Y 130.328,Z 824.842,A -85,B 0,C 180,E1 22783.434,E2 22783.434} C_VEL
LIN {X 0,Y 138.706,Z 818.422,A -85,B 0,C 180,E1 22799.172,E2 22799.172} C_VEL
LIN {X 0,Y 155.124,Z 806.137,A -85,B 0,C 180,E1 22813.094,E2 22813.094} C_VEL
LIN {X 0,Y 177.048,Z 788.182,A -85,B 0,C 180,E1 22823.574,E2 22823.574} C_VEL
LIN {X 0,Y 200.533,Z 765.374,A -85,B 0,C 180,E1 22830.901,E2 22830.901} C_VEL
LIN {X 0,Y 222.521,Z 739.263,A -85,B 0,C 180,E1 22835.908,E2 22835.908} C_VEL
LIN {X 0,Y 231.402,Z 726.983,A -85,B 0,C 180,E1 22837.543,E2 22837.543} C_VEL
LIN {X 0,Y 233.308,Z 716.288,A -85,B 0,C 180,E1 22843.066,E2 22843.066} C_VEL
LIN {X 0,Y 234.237,Z 708.437,A -85,B 0,C 180,E1 22848.82,E2 22848.82} C_VEL
LIN {X 0,Y 234.703,Z 705.186,A -85,B 0,C 180,E1 22852.588,E2 22852.588} C_VEL
LIN {X 0,Y 234.91,Z 703.652,A -85,B 0,C 180,E1 22856.306,E2 22856.306} C_VEL
LIN {X 0,Y 235.197,Z 703.583,A -85,B 0,C 180,E1 22860.001,E2 22860.001} C_VEL
LIN {X 0,Y 235.031,Z 707.4,A -85,B 0,C 180,E1 22865.545,E2 22865.545} C_VEL
LIN {X 0,Y 234.53,Z 716.183,A -85,B 0,C 180,E1 22872.112,E2 22872.112} C_VEL
LIN {X 0,Y 233.563,Z 725.792,A -85,B 0,C 180,E1 22877.03,E2 22877.03} C_VEL
LIN {X 0,Y 231.505,Z 729.937,A -85,B 0,C 180,E1 22877.863,E2 22877.863} C_VEL
LIN {X 0,Y 208.761,Z 760.496,A -85,B 0,C 180,E1 22882.379,E2 22882.379} C_VEL
LIN {X 0,Y 185.181,Z 786.396,A -85,B 0,C 180,E1 22888.736,E2 22888.736} C_VEL
LIN {X 0,Y 163.562,Z 806.814,A -85,B 0,C 180,E1 22897.241,E2 22897.241} C_VEL
LIN {X 0,Y 144.794,Z 823.15,A -85,B 0,C 180,E1 22909.193,E2 22909.193} C_VEL
LIN {X 0,Y 133.396,Z 833.618,A -85,B 0,C 180,E1 22923.001,E2 22923.001} C_VEL
LIN {X 0,Y 128.947,Z 838.997,A -85,B 0,C 180,E1 22936.419,E2 22936.419} C_VEL
LIN {X 0,Y 128.584,Z 840.913,A -85,B 0,C 180,E1 22950.001,E2 22950.001} C_VEL
LIN {X 0,Y 128.959,Z 839.021,A -85,B 0,C 180,E1 22963.582,E2 22963.582} C_VEL
LIN {X 0,Y 133.391,Z 833.656,A -85,B 0,C 180,E1 22977.003,E2 22977.003} C_VEL
LIN {X 0,Y 146.484,Z 821.801,A -85,B 0,C 180,E1 22992.21,E2 22992.21} C_VEL
LIN {X 0,Y 167.365,Z 803.557,A -85,B 0,C 180,E1 23004.508,E2 23004.508} C_VEL
LIN {X 0,Y 191.015,Z 780.551,A -85,B 0,C 180,E1 23013.054,E2 23013.054} C_VEL
LIN {X 0,Y 214.405,Z 753.678,A -85,B 0,C 180,E1 23018.874,E2 23018.874} C_VEL
LIN {X 0,Y 233.022,Z 727.871,A -85,B 0,C 180,E1 23022.384,E2 23022.384} C_VEL
LIN {X 0,Y 234.59,Z 717.954,A -85,B 0,C 180,E1 23026.943,E2 23026.943} C_VEL
LIN {X 0,Y 235.071,Z 709.537,A -85,B 0,C 180,E1 23032.599,E2 23032.599} C_VEL
LIN {X 0,Y 235.178,Z 704.83,A -85,B 0,C 180,E1 23038.155,E2 23038.155} C_VEL
LIN {X 0,Y 235.316,Z 703.824,A -85,B 0,C 180,E1 23039.999,E2 23039.999} C_VEL
LIN {X 0,Y 235.003,Z 703.955,A -85,B 0,C 180,E1 23043.693,E2 23043.693} C_VEL
LIN {X 0,Y 234.47,Z 707.51,A -85,B 0,C 180,E1 23049.897,E2 23049.897} C_VEL
LIN {X 0,Y 233.665,Z 715.049,A -85,B 0,C 180,E1 23055.984,E2 23055.984} C_VEL
LIN {X 0,Y 231.795,Z 726.161,A -85,B 0,C 180,E1 23061.964,E2 23061.964} C_VEL
LIN {X 0,Y 229.711,Z 729.682,A -85,B 0,C 180,E1 23062.666,E2 23062.666} C_VEL
LIN {X 0,Y 208.361,Z 756.954,A -85,B 0,C 180,E1 23067.107,E2 23067.107} C_VEL
LIN {X 0,Y 184.394,Z 781.68,A -85,B 0,C 180,E1 23073.76,E2 23073.76} C_VEL
LIN {X 0,Y 161.282,Z 801.423,A -85,B 0,C 180,E1 23083.318,E2 23083.318} C_VEL
LIN {X 0,Y 142.871,Z 815.386,A -85,B 0,C 180,E1 23096.194,E2 23096.194} C_VEL
LIN {X 0,Y 132.806,Z 822.928,A -85,B 0,C 180,E1 23109.999,E2 23109.999} C_VEL
LIN {X 0,Y 129.05,Z 826.065,A -85,B 0,C 180,E1 23123.261,E2 23123.261} C_VEL
LIN {X 0,Y 128.782,Z 826.323,A -85,B 0,C 180,E1 23132.204,E2 23132.204} C_VEL
LIN {X 0,Y 126.602,Z 826.068,A -85,B 0,C 180,E1 23137.992,E2 23137.992} C_VEL
LIN {X 0,Y 123.766,Z 824.482,A -85,B 0,C 180,E1 23147.707,E2 23147.707} C_VEL
LIN {X 0,Y 123.862,Z 824.253,A -85,B 0,C 180,E1 23147.957,E2 23147.957} C_VEL
LIN {X 0,Y 134.802,Z 816.818,A -85,B 0,C 180,E1 23164.164,E2 23164.164} C_VEL
LIN {X 0,Y 153.783,Z 803.376,A -85,B 0,C 180,E1 23177.594,E2 23177.594} C_VEL
LIN {X 0,Y 176.094,Z 785.455,A -85,B 0,C 180,E1 23186.959,E2 23186.959} C_VEL
LIN {X 0,Y 200.542,Z 761.923,A -85,B 0,C 180,E1 23193.825,E2 23193.825} C_VEL
LIN {X 0,Y 224.08,Z 733.743,A -85,B 0,C 180,E1 23198.617,E2 23198.617} C_VEL
LIN {X 0,Y 226.661,Z 729.831,A -85,B 0,C 180,E1 23199.254,E2 23199.254} C_VEL
LIN {X 0,Y 228.914,Z 718.707,A -85,B 0,C 180,E1 23205.913,E2 23205.913} C_VEL
LIN {X 0,Y 230.175,Z 711.936,A -85,B 0,C 180,E1 23212.442,E2 23212.442} C_VEL
LIN {X 0,Y 230.547,Z 710.308,A -85,B 0,C 180,E1 23216.235,E2 23216.235} C_VEL
LIN {X 0,Y 230.851,Z 710.255,A -85,B 0,C 180,E1 23220.001,E2 23220.001} C_VEL
LIN {X 0,Y 230.393,Z 715.144,A -85,B 0,C 180,E1 23226.604,E2 23226.604} C_VEL
LIN {X 0,Y 229.276,Z 724.959,A -85,B 0,C 180,E1 23233.315,E2 23233.315} C_VEL
LIN {X 0,Y 228.522,Z 729.992,A -85,B 0,C 180,E1 23235.86,E2 23235.86} C_VEL
LIN {X 0,Y 205.791,Z 759.985,A -85,B 0,C 180,E1 23240.277,E2 23240.277} C_VEL
LIN {X 0,Y 180.753,Z 786.509,A -85,B 0,C 180,E1 23246.654,E2 23246.654} C_VEL
LIN {X 0,Y 157.163,Z 807.647,A -85,B 0,C 180,E1 23255.606,E2 23255.606} C_VEL
LIN {X 0,Y 136.937,Z 824.098,A -85,B 0,C 180,E1 23268.442,E2 23268.442} C_VEL
LIN {X 0,Y 124.022,Z 835.267,A -85,B 0,C 180,E1 23285.669,E2 23285.669} C_VEL
LIN {X 0,Y 121.163,Z 838.546,A -85,B 0,C 180,E1 23295.529,E2 23295.529} C_VEL
LIN {X 0,Y 120.674,Z 840.469,A -85,B 0,C 180,E1 23310.001,E2 23310.001} C_VEL
LIN {X 0,Y 121.175,Z 838.57,A -85,B 0,C 180,E1 23324.473,E2 23324.473} C_VEL
LIN {X 0,Y 126.175,Z 833.199,A -85,B 0,C 180,E1 23338.686,E2 23338.686} C_VEL
LIN {X 0,Y 140.521,Z 821.341,A -85,B 0,C 180,E1 23354.456,E2 23354.456} C_VEL
LIN {X 0,Y 162.711,Z 803.081,A -85,B 0,C 180,E1 23366.875,E2 23366.875} C_VEL
LIN {X 0,Y 186.951,Z 780.578,A -85,B 0,C 180,E1 23375.141,E2 23375.141} C_VEL
LIN {X 0,Y 210.45,Z 754.594,A -85,B 0,C 180,E1 23380.693,E2 23380.693} C_VEL
LIN {X 0,Y 228.597,Z 730.165,A -85,B 0,C 180,E1 23384.146,E2 23384.146} C_VEL
LIN {X 0,Y 230.213,Z 718.855,A -85,B 0,C 180,E1 23390.582,E2 23390.582} C_VEL
LIN {X 0,Y 230.745,Z 712.643,A -85,B 0,C 180,E1 23396.237,E2 23396.237} C_VEL
LIN {X 0,Y 230.958,Z 710.492,A -85,B 0,C 180,E1 23399.999,E2 23399.999} C_VEL
LIN {X 0,Y 230.617,Z 710.617,A -85,B 0,C 180,E1 23403.763,E2 23403.763} C_VEL
LIN {X 0,Y 229.863,Z 714.51,A -85,B 0,C 180,E1 23410.263,E2 23410.263} C_VEL
LIN {X 0,Y 228.455,Z 722.289,A -85,B 0,C 180,E1 23416.357,E2 23416.357} C_VEL
LIN {X 0,Y 226.237,Z 730.985,A -85,B 0,C 180,E1 23420.918,E2 23420.918} C_VEL
LIN {X 0,Y 203.34,Z 759.163,A -85,B 0,C 180,E1 23425.467,E2 23425.467} C_VEL
LIN {X 0,Y 178.715,Z 783.341,A -85,B 0,C 180,E1 23432.091,E2 23432.091} C_VEL
LIN {X 0,Y 155.893,Z 801.875,A -85,B 0,C 180,E1 23441.175,E2 23441.175} C_VEL
LIN {X 0,Y 136.284,Z 815.836,A -85,B 0,C 180,E1 23454.319,E2 23454.319} C_VEL
LIN {X 0,Y 125.353,Z 823.374,A -85,B 0,C 180,E1 23468.754,E2 23468.754} C_VEL
LIN {X 0,Y 121.206,Z 826.508,A -85,B 0,C 180,E1 23482.823,E2 23482.823} C_VEL
LIN {X 0,Y 120.89,Z 826.777,A -85,B 0,C 180,E1 23492.172,E2 23492.172} C_VEL
LIN {X 0,Y 123.862,Z 824.253,A -85,B 0,C 180,E1 23507.957,E2 23507.957} C_VEL
LIN {X 0,Y 124.281,Z 822.638,A -85,B 0,C 180,E1 23513.971,E2 23513.971} C_VEL
LIN {X 0,Y 125.27,Z 819.188,A -85,B 0,C 180,E1 23522.963,E2 23522.963} C_VEL
LIN {X 0,Y 126,Z 818.663,A -85,B 0,C 180,E1 23523.882,E2 23523.882} C_VEL
LIN {X 0,Y 146.158,Z 805.515,A -85,B 0,C 180,E1 23538.678,E2 23538.678} C_VEL
LIN {X 0,Y 170.475,Z 787.092,A -85,B 0,C 180,E1 23548.739,E2 23548.739} C_VEL
LIN {X 0,Y 195.468,Z 764.128,A -85,B 0,C 180,E1 23555.521,E2 23555.521} C_VEL
LIN {X 0,Y 219.264,Z 736.875,A -85,B 0,C 180,E1 23560.177,E2 23560.177} C_VEL
LIN {X 0,Y 221.806,Z 733.236,A -85,B 0,C 180,E1 23560.901,E2 23560.901} C_VEL
LIN {X 0,Y 224.337,Z 723.377,A -85,B 0,C 180,E1 23567.331,E2 23567.331} C_VEL
LIN {X 0,Y 225.492,Z 718.612,A -85,B 0,C 180,E1 23572.284,E2 23572.284} C_VEL
LIN {X 0,Y 226.041,Z 716.9,A -85,B 0,C 180,E1 23576.16,E2 23576.16} C_VEL
LIN {X 0,Y 226.385,Z 716.813,A -85,B 0,C 180,E1 23580.001,E2 23580.001} C_VEL
LIN {X 0,Y 225.594,Z 721.858,A -85,B 0,C 180,E1 23586.745,E2 23586.745} C_VEL
LIN {X 0,Y 223.969,Z 731.459,A -85,B 0,C 180,E1 23593.259,E2 23593.259} C_VEL
LIN {X 0,Y 222.995,Z 734.439,A -85,B 0,C 180,E1 23594.573,E2 23594.573} C_VEL
LIN {X 0,Y 199.89,Z 763.067,A -85,B 0,C 180,E1 23598.775,E2 23598.775} C_VEL
LIN {X 0,Y 173.731,Z 789.256,A -85,B 0,C 180,E1 23605.296,E2 23605.296} C_VEL
LIN {X 0,Y 148.128,Z 810.653,A -85,B 0,C 180,E1 23615.147,E2 23615.147} C_VEL
LIN {X 0,Y 127.374,Z 826.243,A -85,B 0,C 180,E1 23629.175,E2 23629.175} C_VEL
LIN {X 0,Y 115.538,Z 835.831,A -85,B 0,C 180,E1 23646.852,E2 23646.852} C_VEL
LIN {X 0,Y 112.476,Z 839.493,A -85,B 0,C 180,E1 23662.265,E2 23662.265} C_VEL
LIN {X 0,Y 112.759,Z 840.025,A -85,B 0,C 180,E1 23670.001,E2 23670.001} C_VEL
LIN {X 0,Y 113.417,Z 838.12,A -85,B 0,C 180,E1 23685.487,E2 23685.487} C_VEL
LIN {X 0,Y 119.091,Z 832.743,A -85,B 0,C 180,E1 23700.568,E2 23700.568} C_VEL
LIN {X 0,Y 135.477,Z 820.392,A -85,B 0,C 180,E1 23717.383,E2 23717.383} C_VEL
LIN {X 0,Y 158.38,Z 802.609,A -85,B 0,C 180,E1 23729.359,E2 23729.359} C_VEL
LIN {X 0,Y 183.424,Z 780.328,A -85,B 0,C 180,E1 23737.391,E2 23737.391} C_VEL
LIN {X 0,Y 207.865,Z 754.125,A -85,B 0,C 180,E1 23742.801,E2 23742.801} C_VEL
LIN {X 0,Y 223.616,Z 733.624,A -85,B 0,C 180,E1 23745.683,E2 23745.683} C_VEL
LIN {X 0,Y 225.564,Z 723.14,A -85,B 0,C 180,E1 23752.285,E2 23752.285} C_VEL
LIN {X 0,Y 226.247,Z 718.165,A -85,B 0,C 180,E1 23757.895,E2 23757.895} C_VEL
LIN {X 0,Y 226.488,Z 717.047,A -85,B 0,C 180,E1 23759.999,E2 23759.999} C_VEL
LIN {X 0,Y 226.095,Z 717.205,A -85,B 0,C 180,E1 23763.839,E2 23763.839} C_VEL
LIN {X 0,Y 225.23,Z 720.168,A -85,B 0,C 180,E1 23769.325,E2 23769.325} C_VEL
LIN {X 0,Y 223.409,Z 727.822,A -85,B 0,C 180,E1 23775.727,E2 23775.727} C_VEL
LIN {X 0,Y 221.498,Z 734.304,A -85,B 0,C 180,E1 23779.356,E2 23779.356} C_VEL
LIN {X 0,Y 196.95,Z 762.851,A -85,B 0,C 180,E1 23784.09,E2 23784.09} C_VEL
LIN {X 0,Y 171.774,Z 786.145,A -85,B 0,C 180,E1 23790.751,E2 23790.751} C_VEL
LIN {X 0,Y 148.365,Z 804.006,A -85,B 0,C 180,E1 23800.058,E2 23800.058} C_VEL
LIN {X 0,Y 128.205,Z 817.38,A -85,B 0,C 180,E1 23813.807,E2 23813.807} C_VEL
LIN {X 0,Y 117.968,Z 823.82,A -85,B 0,C 180,E1 23827.353,E2 23827.353} C_VEL
LIN {X 0,Y 113.353,Z 826.952,A -85,B 0,C 180,E1 23842.323,E2 23842.323} C_VEL
LIN {X 0,Y 113.129,Z 827.349,A -85,B 0,C 180,E1 23849.999,E2 23849.999} C_VEL
LIN {X 0,Y 116.134,Z 824.821,A -85,B 0,C 180,E1 23868.712,E2 23868.712} C_VEL
LIN {X 0,Y 126,Z 818.663,A -85,B 0,C 180,E1 23883.882,E2 23883.882} C_VEL
LIN {X 0,Y 129.849,Z 814.571,A -85,B 0,C 180,E1 23891.336,E2 23891.336} C_VEL
LIN {X 0,Y 135.495,Z 809.459,A -85,B 0,C 180,E1 23898.165,E2 23898.165} C_VEL
LIN {X 0,Y 159.334,Z 793.046,A -85,B 0,C 180,E1 23908.781,E2 23908.781} C_VEL
LIN {X 0,Y 184.472,Z 772.11,A -85,B 0,C 180,E1 23915.932,E2 23915.932} C_VEL
LIN {X 0,Y 209.875,Z 745.689,A -85,B 0,C 180,E1 23921.051,E2 23921.051} C_VEL
LIN {X 0,Y 216.581,Z 737.559,A -85,B 0,C 180,E1 23922.122,E2 23922.122} C_VEL
LIN {X 0,Y 219.42,Z 728.923,A -85,B 0,C 180,E1 23928.055,E2 23928.055} C_VEL
LIN {X 0,Y 220.623,Z 725.175,A -85,B 0,C 180,E1 23932.112,E2 23932.112} C_VEL
LIN {X 0,Y 221.254,Z 723.311,A -85,B 0,C 180,E1 23936.077,E2 23936.077} C_VEL
LIN {X 0,Y 221.631,Z 723.19,A -85,B 0,C 180,E1 23940.001,E2 23940.001} C_VEL
LIN {X 0,Y 220.625,Z 728.507,A -85,B 0,C 180,E1 23946.898,E2 23946.898} C_VEL
LIN {X 0,Y 218.593,Z 737.146,A -85,B 0,C 180,E1 23952.791,E2 23952.791} C_VEL
LIN {X 0,Y 192.514,Z 767.796,A -85,B 0,C 180,E1 23957.528,E2 23957.528} C_VEL
LIN {X 0,Y 165.898,Z 792.601,A -85,B 0,C 180,E1 23964.13,E2 23964.13} C_VEL
LIN {X 0,Y 141.006,Z 811.999,A -85,B 0,C 180,E1 23973.681,E2 23973.681} C_VEL
LIN {X 0,Y 121.286,Z 825.78,A -85,B 0,C 180,E1 23986.642,E2 23986.642} C_VEL
LIN {X 0,Y 108.145,Z 835.377,A -85,B 0,C 180,E1 24005.167,E2 24005.167} C_VEL
LIN {X 0,Y 104.587,Z 839.045,A -85,B 0,C 180,E1 24021.678,E2 24021.678} C_VEL
LIN {X 0,Y 104.842,Z 839.581,A -85,B 0,C 180,E1 24030.002,E2 24030.002} C_VEL
LIN {X 0,Y 105.715,Z 837.671,A -85,B 0,C 180,E1 24046.647,E2 24046.647} C_VEL
LIN {X 0,Y 114.441,Z 830.608,A -85,B 0,C 180,E1 24065.953,E2 24065.953} C_VEL
LIN {X 0,Y 131.183,Z 819.088,A -85,B 0,C 180,E1 24080.813,E2 24080.813} C_VEL
LIN {X 0,Y 155.727,Z 801.017,A -85,B 0,C 180,E1 24092.51,E2 24092.51} C_VEL
LIN {X 0,Y 181.644,Z 778.692,A -85,B 0,C 180,E1 24100.083,E2 24100.083} C_VEL
LIN {X 0,Y 207.158,Z 751.807,A -85,B 0,C 180,E1 24105.227,E2 24105.227} C_VEL
LIN {X 0,Y 218.687,Z 737.326,A -85,B 0,C 180,E1 24107.204,E2 24107.204} C_VEL
LIN {X 0,Y 220.736,Z 728.676,A -85,B 0,C 180,E1 24113.106,E2 24113.106} C_VEL
LIN {X 0,Y 221.737,Z 723.411,A -85,B 0,C 180,E1 24119.999,E2 24119.999} C_VEL
LIN {X 0,Y 221.319,Z 723.602,A -85,B 0,C 180,E1 24123.922,E2 24123.922} C_VEL
LIN {X 0,Y 220.186,Z 727.077,A -85,B 0,C 180,E1 24129.897,E2 24129.897} C_VEL
LIN {X 0,Y 217.761,Z 734.923,A -85,B 0,C 180,E1 24136.146,E2 24136.146} C_VEL
LIN {X 0,Y 216.863,Z 737.412,A -85,B 0,C 180,E1 24137.683,E2 24137.683} C_VEL
LIN {X 0,Y 192.248,Z 764.899,A -85,B 0,C 180,E1 24142.273,E2 24142.273} C_VEL
LIN {X 0,Y 166.374,Z 787.78,A -85,B 0,C 180,E1 24148.846,E2 24148.846} C_VEL
LIN {X 0,Y 140.907,Z 806.137,A -85,B 0,C 180,E1 24158.828,E2 24158.828} C_VEL
LIN {X 0,Y 121.841,Z 817.83,A -85,B 0,C 180,E1 24171.586,E2 24171.586} C_VEL
LIN {X 0,Y 110.677,Z 824.265,A -85,B 0,C 180,E1 24185.769,E2 24185.769} C_VEL
LIN {X 0,Y 105.519,Z 827.396,A -85,B 0,C 180,E1 24201.749,E2 24201.749} C_VEL
LIN {X 0,Y 105.247,Z 827.791,A -85,B 0,C 180,E1 24209.998,E2 24209.998} C_VEL
LIN {X 0,Y 107.306,Z 826.179,A -85,B 0,C 180,E1 24226.39,E2 24226.39} C_VEL
LIN {X 0,Y 118.874,Z 819.446,A -85,B 0,C 180,E1 24245.434,E2 24245.434} C_VEL
LIN {X 0,Y 135.495,Z 809.459,A -85,B 0,C 180,E1 24258.165,E2 24258.165} C_VEL
LIN {X 0,Y 142.488,Z 803.541,A -85,B 0,C 180,E1 24264.337,E2 24264.337} C_VEL
LIN {X 0,Y 149.379,Z 797.737,A -85,B 0,C 180,E1 24269.234,E2 24269.234} C_VEL
LIN {X 0,Y 150.79,Z 796.773,A -85,B 0,C 180,E1 24269.761,E2 24269.761} C_VEL
LIN {X 0,Y 178.17,Z 775.468,A -85,B 0,C 180,E1 24277.51,E2 24277.51} C_VEL
LIN {X 0,Y 204.507,Z 749.488,A -85,B 0,C 180,E1 24282.646,E2 24282.646} C_VEL
LIN {X 0,Y 211.418,Z 741.561,A -85,B 0,C 180,E1 24283.72,E2 24283.72} C_VEL
LIN {X 0,Y 213.959,Z 735.66,A -85,B 0,C 180,E1 24287.745,E2 24287.745} C_VEL
LIN {X 0,Y 215.467,Z 731.582,A -85,B 0,C 180,E1 24291.922,E2 24291.922} C_VEL
LIN {X 0,Y 216.308,Z 729.634,A -85,B 0,C 180,E1 24295.987,E2 24295.987} C_VEL
LIN {X 0,Y 216.741,Z 729.492,A -85,B 0,C 180,E1 24300.001,E2 24300.001} C_VEL
LIN {X 0,Y 215.506,Z 734.355,A -85,B 0,C 180,E1 24306.514,E2 24306.514} C_VEL
LIN {X 0,Y 213.732,Z 740.647,A -85,B 0,C 180,E1 24311.121,E2 24311.121} C_VEL
LIN {X 0,Y 188.54,Z 768.938,A -85,B 0,C 180,E1 24315.499,E2 24315.499} C_VEL
LIN {X 0,Y 161.01,Z 793.492,A -85,B 0,C 180,E1 24321.974,E2 24321.974} C_VEL
LIN {X 0,Y 133.987,Z 813.346,A -85,B 0,C 180,E1 24332.061,E2 24332.061} C_VEL
LIN {X 0,Y 111.688,Z 827.754,A -85,B 0,C 180,E1 24347.33,E2 24347.33} C_VEL
LIN {X 0,Y 100.012,Z 835.545,A -85,B 0,C 180,E1 24365.269,E2 24365.269} C_VEL
LIN {X 0,Y 96.703,Z 838.597,A -85,B 0,C 180,E1 24380.994,E2 24380.994} C_VEL
LIN {X 0,Y 96.923,Z 839.136,A -85,B 0,C 180,E1 24390.002,E2 24390.002} C_VEL
LIN {X 0,Y 98.033,Z 837.219,A -85,B 0,C 180,E1 24407.994,E2 24407.994} C_VEL
LIN {X 0,Y 107.73,Z 830.28,A -85,B 0,C 180,E1 24428.261,E2 24428.261} C_VEL
LIN {X 0,Y 126.139,Z 818.626,A -85,B 0,C 180,E1 24443.709,E2 24443.709} C_VEL
LIN {X 0,Y 150.656,Z 801.661,A -85,B 0,C 180,E1 24454.755,E2 24454.755} C_VEL
LIN {X 0,Y 178.53,Z 778.659,A -85,B 0,C 180,E1 24462.436,E2 24462.436} C_VEL
LIN {X 0,Y 204.263,Z 752.402,A -85,B 0,C 180,E1 24467.266,E2 24467.266} C_VEL
LIN {X 0,Y 213.803,Z 740.849,A -85,B 0,C 180,E1 24468.866,E2 24468.866} C_VEL
LIN {X 0,Y 215.9,Z 733.174,A -85,B 0,C 180,E1 24474.902,E2 24474.902} C_VEL
LIN {X 0,Y 216.839,Z 729.703,A -85,B 0,C 180,E1 24479.999,E2 24479.999} C_VEL
LIN {X 0,Y 216.365,Z 729.909,A -85,B 0,C 180,E1 24484.012,E2 24484.012} C_VEL
LIN {X 0,Y 215.061,Z 733.187,A -85,B 0,C 180,E1 24489.725,E2 24489.725} C_VEL
LIN {X 0,Y 212.216,Z 740.589,A -85,B 0,C 180,E1 24495.769,E2 24495.769} C_VEL
LIN {X 0,Y 205.874,Z 748.199,A -85,B 0,C 180,E1 24497.046,E2 24497.046} C_VEL
LIN {X 0,Y 179.708,Z 774.275,A -85,B 0,C 180,E1 24502.063,E2 24502.063} C_VEL
LIN {X 0,Y 152.257,Z 795.91,A -85,B 0,C 180,E1 24509.656,E2 24509.656} C_VEL
LIN {X 0,Y 126.199,Z 812.4,A -85,B 0,C 180,E1 24521.489,E2 24521.489} C_VEL
LIN {X 0,Y 107.973,Z 822.376,A -85,B 0,C 180,E1 24537.274,E2 24537.274} C_VEL
LIN {X 0,Y 99.671,Z 826.67,A -85,B 0,C 180,E1 24552.312,E2 24552.312} C_VEL
LIN {X 0,Y 97.35,Z 828.234,A -85,B 0,C 180,E1 24569.998,E2 24569.998} C_VEL
LIN {X 0,Y 99.711,Z 826.625,A -85,B 0,C 180,E1 24587.678,E2 24587.678} C_VEL
LIN {X 0,Y 112.108,Z 820.096,A -85,B 0,C 180,E1 24607.424,E2 24607.424} C_VEL
LIN {X 0,Y 133.584,Z 807.945,A -85,B 0,C 180,E1 24622.501,E2 24622.501} C_VEL
LIN {X 0,Y 150.79,Z 796.773,A -85,B 0,C 180,E1 24629.761,E2 24629.761} C_VEL
LIN {X 0,Y 155.867,Z 792.948,A -85,B 0,C 180,E1 24632.01,E2 24632.01} C_VEL
LIN {X 0,Y 168.121,Z 781.813,A -85,B 0,C 180,E1 24638.275,E2 24638.275} C_VEL
LIN {X 0,Y 169.586,Z 780.6,A -85,B 0,C 180,E1 24638.651,E2 24638.651} C_VEL
LIN {X 0,Y 196.212,Z 756.404,A -85,B 0,C 180,E1 24643.82,E2 24643.82} C_VEL
LIN {X 0,Y 206.69,Z 745.154,A -85,B 0,C 180,E1 24645.436,E2 24645.436} C_VEL
LIN {X 0,Y 209.529,Z 739.247,A -85,B 0,C 180,E1 24650.096,E2 24650.096} C_VEL
LIN {X 0,Y 211.204,Z 735.86,A -85,B 0,C 180,E1 24655.89,E2 24655.89} C_VEL
LIN {X 0,Y 211.68,Z 735.654,A -85,B 0,C 180,E1 24660.001,E2 24660.001} C_VEL
LIN {X 0,Y 210.012,Z 740.805,A -85,B 0,C 180,E1 24666.685,E2 24666.685} C_VEL
LIN {X 0,Y 208.322,Z 745.084,A -85,B 0,C 180,E1 24669.672,E2 24669.672} C_VEL
LIN {X 0,Y 181.207,Z 773.548,A -85,B 0,C 180,E1 24674.051,E2 24674.051} C_VEL
LIN {X 0,Y 151.807,Z 797.804,A -85,B 0,C 180,E1 24680.978,E2 24680.978} C_VEL
LIN {X 0,Y 124.396,Z 816.236,A -85,B 0,C 180,E1 24691.574,E2 24691.574} C_VEL
LIN {X 0,Y 102.632,Z 829.06,A -85,B 0,C 180,E1 24707.526,E2 24707.526} C_VEL
LIN {X 0,Y 91.288,Z 836.085,A -85,B 0,C 180,E1 24727.14,E2 24727.14} C_VEL
LIN {X 0,Y 88.857,Z 838.151,A -85,B 0,C 180,E1 24740.191,E2 24740.191} C_VEL
LIN {X 0,Y 89,Z 838.692,A -85,B 0,C 180,E1 24750.002,E2 24750.002} C_VEL
LIN {X 0,Y 90.412,Z 836.768,A -85,B 0,C 180,E1 24769.57,E2 24769.57} C_VEL
LIN {X 0,Y 100.676,Z 830.295,A -85,B 0,C 180,E1 24790.191,E2 24790.191} C_VEL
LIN {X 0,Y 121.779,Z 817.953,A -85,B 0,C 180,E1 24807.022,E2 24807.022} C_VEL
LIN {X 0,Y 149.542,Z 799.57,A -85,B 0,C 180,E1 24818.349,E2 24818.349} C_VEL
LIN {X 0,Y 178.156,Z 776.461,A -85,B 0,C 180,E1 24825.356,E2 24825.356} C_VEL
LIN {X 0,Y 205.8,Z 748.372,A -85,B 0,C 180,E1 24829.947,E2 24829.947} C_VEL
LIN {X 0,Y 208.963,Z 744.397,A -85,B 0,C 180,E1 24830.617,E2 24830.617} C_VEL
LIN {X 0,Y 210.925,Z 738.484,A -85,B 0,C 180,E1 24835.883,E2 24835.883} C_VEL
LIN {X 0,Y 211.785,Z 735.857,A -85,B 0,C 180,E1 24839.999,E2 24839.999} C_VEL
LIN {X 0,Y 211.264,Z 736.126,A -85,B 0,C 180,E1 24844.109,E2 24844.109} C_VEL
LIN {X 0,Y 209.549,Z 739.591,A -85,B 0,C 180,E1 24849.984,E2 24849.984} C_VEL
LIN {X 0,Y 206.766,Z 745.338,A -85,B 0,C 180,E1 24854.485,E2 24854.485} C_VEL
LIN {X 0,Y 180.164,Z 771.886,A -85,B 0,C 180,E1 24859.014,E2 24859.014} C_VEL
LIN {X 0,Y 153.132,Z 793.103,A -85,B 0,C 180,E1 24865.548,E2 24865.548} C_VEL
LIN {X 0,Y 126.229,Z 809.987,A -85,B 0,C 180,E1 24875.868,E2 24875.868} C_VEL
LIN {X 0,Y 105.805,Z 820.636,A -85,B 0,C 180,E1 24889.912,E2 24889.912} C_VEL
LIN {X 0,Y 92.132,Z 827.115,A -85,B 0,C 180,E1 24910.81,E2 24910.81} C_VEL
LIN {X 0,Y 89.46,Z 828.677,A -85,B 0,C 180,E1 24929.998,E2 24929.998} C_VEL
LIN {X 0,Y 92.173,Z 827.071,A -85,B 0,C 180,E1 24949.177,E2 24949.177} C_VEL
LIN {X 0,Y 105.857,Z 820.545,A -85,B 0,C 180,E1 24970.061,E2 24970.061} C_VEL
LIN {X 0,Y 128.872,Z 808.397,A -85,B 0,C 180,E1 24985.323,E2 24985.323} C_VEL
LIN {X 0,Y 156.275,Z 790.798,A -85,B 0,C 180,E1 24995.267,E2 24995.267} C_VEL
LIN {X 0,Y 169.586,Z 780.6,A -85,B 0,C 180,E1 24998.651,E2 24998.651} C_VEL
LIN {X 0,Y 179.717,Z 771.371,A -85,B 0,C 180,E1 25002.254,E2 25002.254} C_VEL
LIN {X 0,Y 189.802,Z 761.231,A -85,B 0,C 180,E1 25005.397,E2 25005.397} C_VEL
LIN {X 0,Y 201.858,Z 748.88,A -85,B 0,C 180,E1 25007.178,E2 25007.178} C_VEL
LIN {X 0,Y 204.634,Z 744.06,A -85,B 0,C 180,E1 25011.586,E2 25011.586} C_VEL
LIN {X 0,Y 205.845,Z 741.863,A -85,B 0,C 180,E1 25015.783,E2 25015.783} C_VEL
LIN {X 0,Y 206.382,Z 741.647,A -85,B 0,C 180,E1 25020.001,E2 25020.001} C_VEL
LIN {X 0,Y 204.628,Z 746.416,A -85,B 0,C 180,E1 25026.254,E2 25026.254} C_VEL
LIN {X 0,Y 203.946,Z 748.098,A -85,B 0,C 180,E1 25027.668,E2 25027.668} C_VEL
LIN {X 0,Y 176.299,Z 775.765,A -85,B 0,C 180,E1 25032.072,E2 25032.072} C_VEL
LIN {X 0,Y 147.771,Z 798.227,A -85,B 0,C 180,E1 25038.379,E2 25038.379} C_VEL
LIN {X 0,Y 120.31,Z 815.771,A -85,B 0,C 180,E1 25048.249,E2 25048.249} C_VEL
LIN {X 0,Y 96.749,Z 828.599,A -85,B 0,C 180,E1 25064.249,E2 25064.249} C_VEL
LIN {X 0,Y 84.229,Z 835.444,A -85,B 0,C 180,E1 25083.993,E2 25083.993} C_VEL
LIN {X 0,Y 80.997,Z 837.702,A -85,B 0,C 180,E1 25099.228,E2 25099.228} C_VEL
LIN {X 0,Y 81.076,Z 838.247,A -85,B 0,C 180,E1 25110.002,E2 25110.002} C_VEL
LIN {X 0,Y 82.862,Z 836.316,A -85,B 0,C 180,E1 25131.437,E2 25131.437} C_VEL
LIN {X 0,Y 96.8,Z 828.638,A -85,B 0,C 180,E1 25155.78,E2 25155.78} C_VEL
LIN {X 0,Y 120.317,Z 815.866,A -85,B 0,C 180,E1 25171.751,E2 25171.751} C_VEL
LIN {X 0,Y 150.146,Z 796.71,A -85,B 0,C 180,E1 25182.268,E2 25182.268} C_VEL
LIN {X 0,Y 181.198,Z 771.551,A -85,B 0,C 180,E1 25188.804,E2 25188.804} C_VEL
LIN {X 0,Y 204.087,Z 748.212,A -85,B 0,C 180,E1 25192.327,E2 25192.327} C_VEL
LIN {X 0,Y 205.998,Z 743.02,A -85,B 0,C 180,E1 25197.893,E2 25197.893} C_VEL
LIN {X 0,Y 206.479,Z 741.84,A -85,B 0,C 180,E1 25199.999,E2 25199.999} C_VEL
LIN {X 0,Y 205.321,Z 743.047,A -85,B 0,C 180,E1 25206.349,E2 25206.349} C_VEL
LIN {X 0,Y 202.819,Z 747.8,A -85,B 0,C 180,E1 25212.065,E2 25212.065} C_VEL
LIN {X 0,Y 200.493,Z 750.609,A -85,B 0,C 180,E1 25212.923,E2 25212.923} C_VEL
LIN {X 0,Y 172.404,Z 776.883,A -85,B 0,C 180,E1 25217.586,E2 25217.586} C_VEL
LIN {X 0,Y 143.311,Z 797.884,A -85,B 0,C 180,E1 25224.677,E2 25224.677} C_VEL
LIN {X 0,Y 115.899,Z 813.458,A -85,B 0,C 180,E1 25235.753,E2 25235.753} C_VEL
LIN {X 0,Y 95.954,Z 822.843,A -85,B 0,C 180,E1 25250.862,E2 25250.862} C_VEL
LIN {X 0,Y 84.668,Z 827.561,A -85,B 0,C 180,E1 25269.042,E2 25269.042} C_VEL
LIN {X 0,Y 81.561,Z 829.12,A -85,B 0,C 180,E1 25289.998,E2 25289.998} C_VEL
LIN {X 0,Y 84.709,Z 827.517,A -85,B 0,C 180,E1 25310.943,E2 25310.943} C_VEL
